// TIA Portal V17 export
// export: Created 2025-03-05T08:01:38.605309Z, ExportSetting WithDefaults, DisplayName Totally Integrated Automation Portal, DisplayVersion V17 Update 8, DisplayName TIA Portal Openness, DisplayVersion V17 Update 8, DisplayName TIA Portal Version Control Interface, DisplayVersion V17, DisplayName SINAMICS Startdrive Advanced, DisplayVersion V17 SP2, DisplayName SINAMICS Startdrive G110M, G120, G120C, G120D, G120P, G115D, DisplayVersion V17 SP2, DisplayName SINAMICS Startdrive G130, G150, S120, S150, SINAMICS MV, S210, DisplayVersion V17 SP2, DisplayName STEP 7 Professional, DisplayVersion V17 Update 8, DisplayName SINUMERIK ONE STEP 7 Toolbox, DisplayVersion V17 Update 12, DisplayName SINUMERIK 840D sl STEP 7 Toolbox, DisplayVersion V17 Update 12, DisplayName STEP 7 Safety, DisplayVersion V17 Update 6, DisplayName WinCC Advanced, DisplayVersion V17 Update 8
FUNCTION "FC7217_TRADES_CALL" : Void   // FC7217, LAD
{ S7_Optimized_Access := 'FALSE' }
AUTHOR : ETXETAR
VERSION : 1.0
// stored: AutoNumber false, IsIECCheckEnabled false, SetENOAutomatically false, UDAEnableTagReadback false
   VAR CONSTANT
      FC_NUMBER : DInt := 7217;
   END_VAR
   VAR_TEMP   // added for the SCL form of the ladder/FBD networks
      _w1 : Bool;
      _w2 : Bool;
      _w3 : Bool;
      _w4 : Bool;
      _w5 : Bool;
      _w6 : Bool;
      _w7 : Bool;
      _w8 : Bool;
      _w9 : Bool;
      _w10 : Bool;
      _w11 : Bool;
      _w12 : Bool;
      _w13 : Bool;
      _w14 : Bool;
      _w15 : Bool;
      _w16 : Bool;
   END_VAR
BEGIN

REGION Network 1: GENERAL CONDITIONS
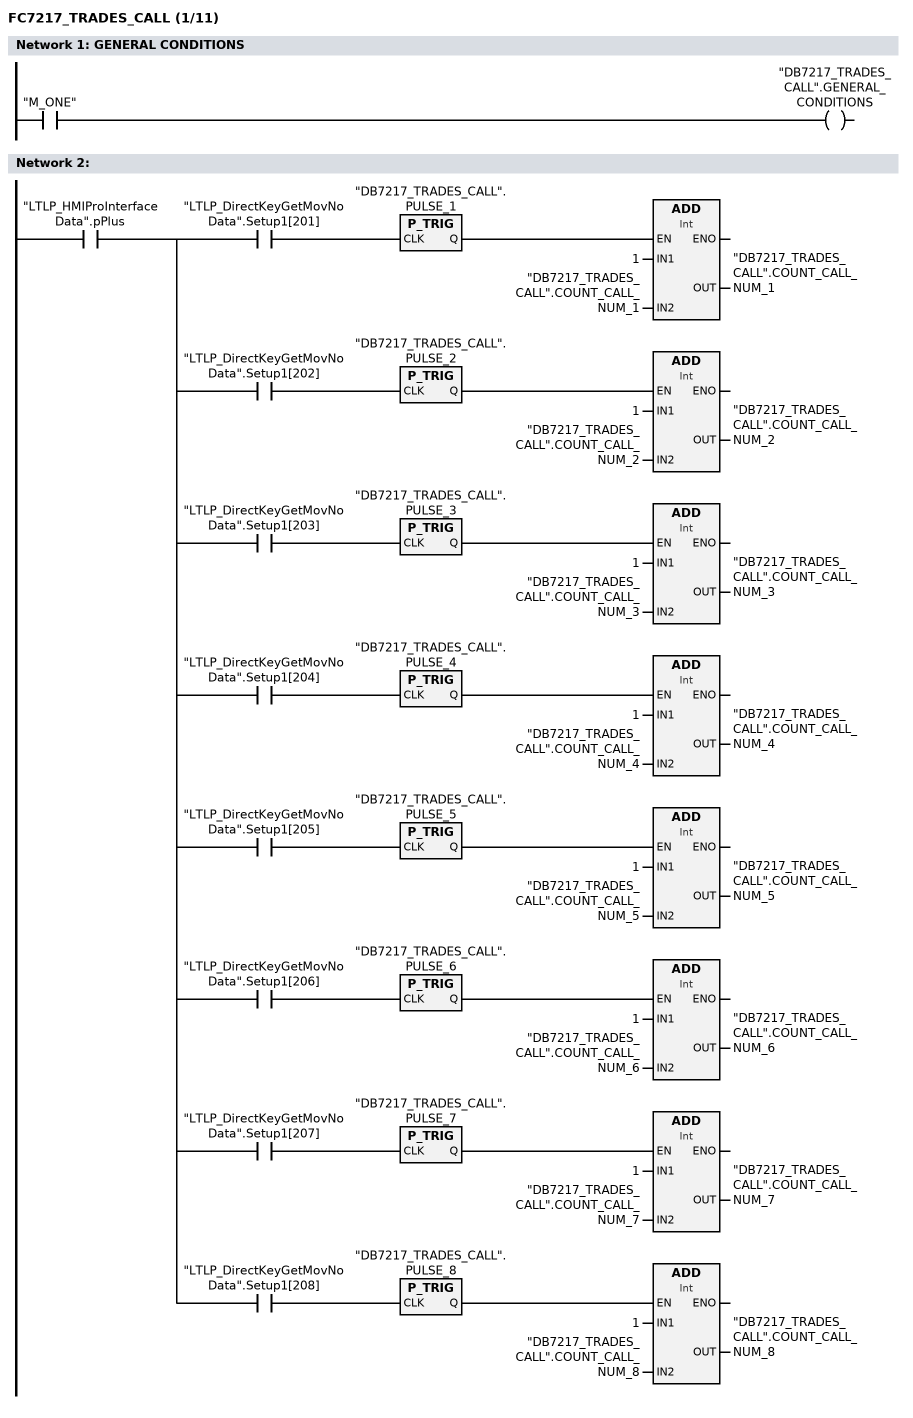
   RUNG wire#powerrail
      Contact( "M_ONE" )
      Coil( "DB7217_TRADES_CALL".GENERAL_CONDITIONS )
   END_RUNG
   // the same network as SCL:
   "DB7217_TRADES_CALL".GENERAL_CONDITIONS := "M_ONE";
END_REGION

REGION Network 2
   RUNG wire#powerrail
      Contact( "LTLP_HMIProInterfaceData".pPlus )
      wire#w1
      Contact( "LTLP_DirectKeyGetMovNoData".Setup1[201] )
      P_Trig( "DB7217_TRADES_CALL".PULSE_1 )
      { S7_Templates := "SrcType := Int"; S7_GenerateENO := "TRUE" } Add(in1 := 1, in2 := "DB7217_TRADES_CALL".COUNT_CALL_NUM_1, out => "DB7217_TRADES_CALL".COUNT_CALL_NUM_1)
   END_RUNG
   RUNG wire#w1
      Contact( "LTLP_DirectKeyGetMovNoData".Setup1[202] )
      P_Trig( "DB7217_TRADES_CALL".PULSE_2 )
      { S7_Templates := "SrcType := Int"; S7_GenerateENO := "TRUE" } Add(in1 := 1, in2 := "DB7217_TRADES_CALL".COUNT_CALL_NUM_2, out => "DB7217_TRADES_CALL".COUNT_CALL_NUM_2)
   END_RUNG
   RUNG wire#w1
      Contact( "LTLP_DirectKeyGetMovNoData".Setup1[203] )
      P_Trig( "DB7217_TRADES_CALL".PULSE_3 )
      { S7_Templates := "SrcType := Int"; S7_GenerateENO := "TRUE" } Add(in1 := 1, in2 := "DB7217_TRADES_CALL".COUNT_CALL_NUM_3, out => "DB7217_TRADES_CALL".COUNT_CALL_NUM_3)
   END_RUNG
   RUNG wire#w1
      Contact( "LTLP_DirectKeyGetMovNoData".Setup1[204] )
      P_Trig( "DB7217_TRADES_CALL".PULSE_4 )
      { S7_Templates := "SrcType := Int"; S7_GenerateENO := "TRUE" } Add(in1 := 1, in2 := "DB7217_TRADES_CALL".COUNT_CALL_NUM_4, out => "DB7217_TRADES_CALL".COUNT_CALL_NUM_4)
   END_RUNG
   RUNG wire#w1
      Contact( "LTLP_DirectKeyGetMovNoData".Setup1[205] )
      P_Trig( "DB7217_TRADES_CALL".PULSE_5 )
      { S7_Templates := "SrcType := Int"; S7_GenerateENO := "TRUE" } Add(in1 := 1, in2 := "DB7217_TRADES_CALL".COUNT_CALL_NUM_5, out => "DB7217_TRADES_CALL".COUNT_CALL_NUM_5)
   END_RUNG
   RUNG wire#w1
      Contact( "LTLP_DirectKeyGetMovNoData".Setup1[206] )
      P_Trig( "DB7217_TRADES_CALL".PULSE_6 )
      { S7_Templates := "SrcType := Int"; S7_GenerateENO := "TRUE" } Add(in1 := 1, in2 := "DB7217_TRADES_CALL".COUNT_CALL_NUM_6, out => "DB7217_TRADES_CALL".COUNT_CALL_NUM_6)
   END_RUNG
   RUNG wire#w1
      Contact( "LTLP_DirectKeyGetMovNoData".Setup1[207] )
      P_Trig( "DB7217_TRADES_CALL".PULSE_7 )
      { S7_Templates := "SrcType := Int"; S7_GenerateENO := "TRUE" } Add(in1 := 1, in2 := "DB7217_TRADES_CALL".COUNT_CALL_NUM_7, out => "DB7217_TRADES_CALL".COUNT_CALL_NUM_7)
   END_RUNG
   RUNG wire#w1
      Contact( "LTLP_DirectKeyGetMovNoData".Setup1[208] )
      P_Trig( "DB7217_TRADES_CALL".PULSE_8 )
      { S7_Templates := "SrcType := Int"; S7_GenerateENO := "TRUE" } Add(in1 := 1, in2 := "DB7217_TRADES_CALL".COUNT_CALL_NUM_8, out => "DB7217_TRADES_CALL".COUNT_CALL_NUM_8)
   END_RUNG
   // the same network as SCL:
   #_w1 := "LTLP_HMIProInterfaceData".pPlus AND "LTLP_DirectKeyGetMovNoData".Setup1[201];
   #_w2 := #_w1 AND NOT "DB7217_TRADES_CALL".PULSE_1;   // rising edge
   "DB7217_TRADES_CALL".PULSE_1 := #_w1;
   IF #_w2 THEN "DB7217_TRADES_CALL".COUNT_CALL_NUM_1 := 1 + "DB7217_TRADES_CALL".COUNT_CALL_NUM_1; END_IF;
   #_w3 := "LTLP_HMIProInterfaceData".pPlus AND "LTLP_DirectKeyGetMovNoData".Setup1[202];
   #_w4 := #_w3 AND NOT "DB7217_TRADES_CALL".PULSE_2;   // rising edge
   "DB7217_TRADES_CALL".PULSE_2 := #_w3;
   IF #_w4 THEN "DB7217_TRADES_CALL".COUNT_CALL_NUM_2 := 1 + "DB7217_TRADES_CALL".COUNT_CALL_NUM_2; END_IF;
   #_w5 := "LTLP_HMIProInterfaceData".pPlus AND "LTLP_DirectKeyGetMovNoData".Setup1[203];
   #_w6 := #_w5 AND NOT "DB7217_TRADES_CALL".PULSE_3;   // rising edge
   "DB7217_TRADES_CALL".PULSE_3 := #_w5;
   IF #_w6 THEN "DB7217_TRADES_CALL".COUNT_CALL_NUM_3 := 1 + "DB7217_TRADES_CALL".COUNT_CALL_NUM_3; END_IF;
   #_w7 := "LTLP_HMIProInterfaceData".pPlus AND "LTLP_DirectKeyGetMovNoData".Setup1[204];
   #_w8 := #_w7 AND NOT "DB7217_TRADES_CALL".PULSE_4;   // rising edge
   "DB7217_TRADES_CALL".PULSE_4 := #_w7;
   IF #_w8 THEN "DB7217_TRADES_CALL".COUNT_CALL_NUM_4 := 1 + "DB7217_TRADES_CALL".COUNT_CALL_NUM_4; END_IF;
   #_w9 := "LTLP_HMIProInterfaceData".pPlus AND "LTLP_DirectKeyGetMovNoData".Setup1[205];
   #_w10 := #_w9 AND NOT "DB7217_TRADES_CALL".PULSE_5;   // rising edge
   "DB7217_TRADES_CALL".PULSE_5 := #_w9;
   IF #_w10 THEN "DB7217_TRADES_CALL".COUNT_CALL_NUM_5 := 1 + "DB7217_TRADES_CALL".COUNT_CALL_NUM_5; END_IF;
   #_w11 := "LTLP_HMIProInterfaceData".pPlus AND "LTLP_DirectKeyGetMovNoData".Setup1[206];
   #_w12 := #_w11 AND NOT "DB7217_TRADES_CALL".PULSE_6;   // rising edge
   "DB7217_TRADES_CALL".PULSE_6 := #_w11;
   IF #_w12 THEN "DB7217_TRADES_CALL".COUNT_CALL_NUM_6 := 1 + "DB7217_TRADES_CALL".COUNT_CALL_NUM_6; END_IF;
   #_w13 := "LTLP_HMIProInterfaceData".pPlus AND "LTLP_DirectKeyGetMovNoData".Setup1[207];
   #_w14 := #_w13 AND NOT "DB7217_TRADES_CALL".PULSE_7;   // rising edge
   "DB7217_TRADES_CALL".PULSE_7 := #_w13;
   IF #_w14 THEN "DB7217_TRADES_CALL".COUNT_CALL_NUM_7 := 1 + "DB7217_TRADES_CALL".COUNT_CALL_NUM_7; END_IF;
   #_w15 := "LTLP_HMIProInterfaceData".pPlus AND "LTLP_DirectKeyGetMovNoData".Setup1[208];
   #_w16 := #_w15 AND NOT "DB7217_TRADES_CALL".PULSE_8;   // rising edge
   "DB7217_TRADES_CALL".PULSE_8 := #_w15;
   IF #_w16 THEN "DB7217_TRADES_CALL".COUNT_CALL_NUM_8 := 1 + "DB7217_TRADES_CALL".COUNT_CALL_NUM_8; END_IF;
END_REGION

REGION Network 3: CALL 1 AUX
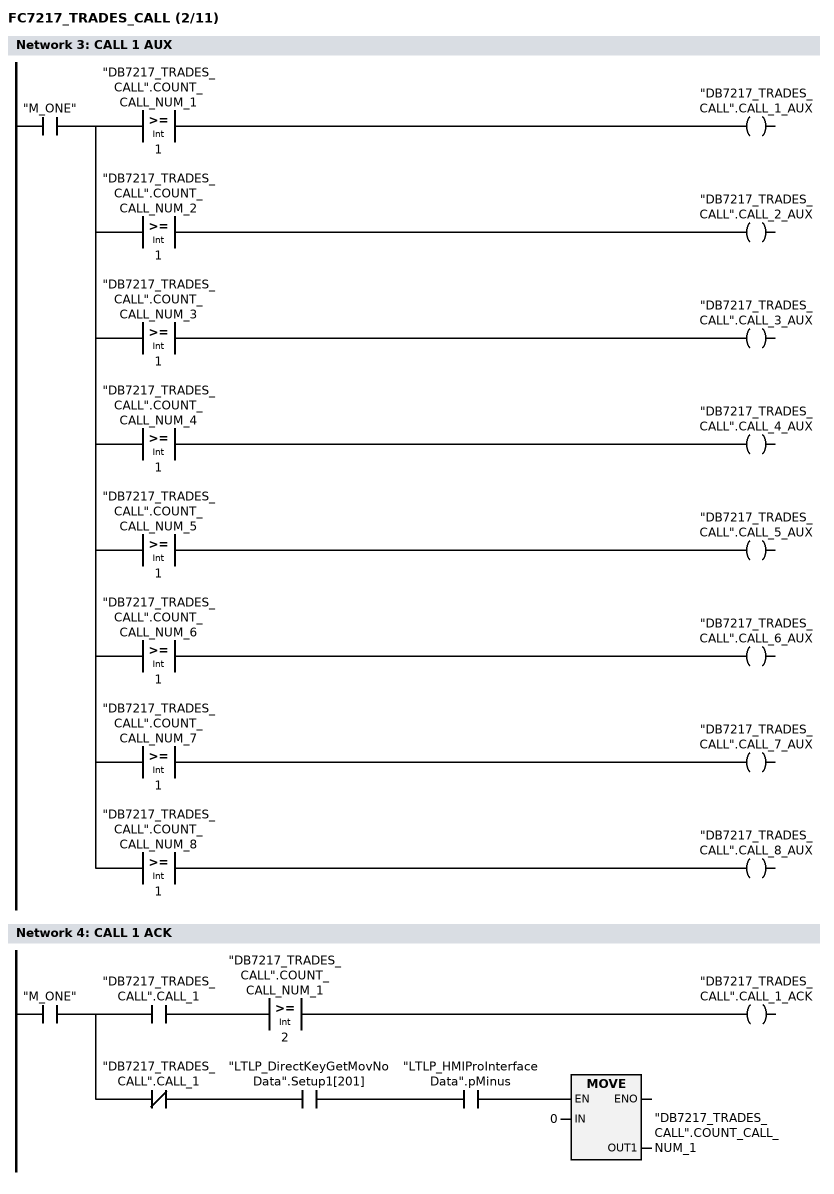
   RUNG wire#powerrail
      Contact( "M_ONE" )
      wire#w1
      { S7_Templates := "SrcType := Int" } GE_Contact(in1 := "DB7217_TRADES_CALL".COUNT_CALL_NUM_1, in2 := 1)
      Coil( "DB7217_TRADES_CALL".CALL_1_AUX )
   END_RUNG
   RUNG wire#w1
      { S7_Templates := "SrcType := Int" } GE_Contact(in1 := "DB7217_TRADES_CALL".COUNT_CALL_NUM_2, in2 := 1)
      Coil( "DB7217_TRADES_CALL".CALL_2_AUX )
   END_RUNG
   RUNG wire#w1
      { S7_Templates := "SrcType := Int" } GE_Contact(in1 := "DB7217_TRADES_CALL".COUNT_CALL_NUM_3, in2 := 1)
      Coil( "DB7217_TRADES_CALL".CALL_3_AUX )
   END_RUNG
   RUNG wire#w1
      { S7_Templates := "SrcType := Int" } GE_Contact(in1 := "DB7217_TRADES_CALL".COUNT_CALL_NUM_4, in2 := 1)
      Coil( "DB7217_TRADES_CALL".CALL_4_AUX )
   END_RUNG
   RUNG wire#w1
      { S7_Templates := "SrcType := Int" } GE_Contact(in1 := "DB7217_TRADES_CALL".COUNT_CALL_NUM_5, in2 := 1)
      Coil( "DB7217_TRADES_CALL".CALL_5_AUX )
   END_RUNG
   RUNG wire#w1
      { S7_Templates := "SrcType := Int" } GE_Contact(in1 := "DB7217_TRADES_CALL".COUNT_CALL_NUM_6, in2 := 1)
      Coil( "DB7217_TRADES_CALL".CALL_6_AUX )
   END_RUNG
   RUNG wire#w1
      { S7_Templates := "SrcType := Int" } GE_Contact(in1 := "DB7217_TRADES_CALL".COUNT_CALL_NUM_7, in2 := 1)
      Coil( "DB7217_TRADES_CALL".CALL_7_AUX )
   END_RUNG
   RUNG wire#w1
      { S7_Templates := "SrcType := Int" } GE_Contact(in1 := "DB7217_TRADES_CALL".COUNT_CALL_NUM_8, in2 := 1)
      Coil( "DB7217_TRADES_CALL".CALL_8_AUX )
   END_RUNG
   // the same network as SCL:
   "DB7217_TRADES_CALL".CALL_1_AUX := "M_ONE" AND ("DB7217_TRADES_CALL".COUNT_CALL_NUM_1 >= 1);
   "DB7217_TRADES_CALL".CALL_2_AUX := "M_ONE" AND ("DB7217_TRADES_CALL".COUNT_CALL_NUM_2 >= 1);
   "DB7217_TRADES_CALL".CALL_3_AUX := "M_ONE" AND ("DB7217_TRADES_CALL".COUNT_CALL_NUM_3 >= 1);
   "DB7217_TRADES_CALL".CALL_4_AUX := "M_ONE" AND ("DB7217_TRADES_CALL".COUNT_CALL_NUM_4 >= 1);
   "DB7217_TRADES_CALL".CALL_5_AUX := "M_ONE" AND ("DB7217_TRADES_CALL".COUNT_CALL_NUM_5 >= 1);
   "DB7217_TRADES_CALL".CALL_6_AUX := "M_ONE" AND ("DB7217_TRADES_CALL".COUNT_CALL_NUM_6 >= 1);
   "DB7217_TRADES_CALL".CALL_7_AUX := "M_ONE" AND ("DB7217_TRADES_CALL".COUNT_CALL_NUM_7 >= 1);
   "DB7217_TRADES_CALL".CALL_8_AUX := "M_ONE" AND ("DB7217_TRADES_CALL".COUNT_CALL_NUM_8 >= 1);
END_REGION

REGION Network 4: CALL 1 ACK
   RUNG wire#powerrail
      Contact( "M_ONE" )
      wire#w1
      Contact( "DB7217_TRADES_CALL".CALL_1 )
      { S7_Templates := "SrcType := Int" } GE_Contact(in1 := "DB7217_TRADES_CALL".COUNT_CALL_NUM_1, in2 := 2)
      Coil( "DB7217_TRADES_CALL".CALL_1_ACK )
   END_RUNG
   RUNG wire#w1
      I_Contact( "DB7217_TRADES_CALL".CALL_1 )
      Contact( "LTLP_DirectKeyGetMovNoData".Setup1[201] )
      Contact( "LTLP_HMIProInterfaceData".pMinus )
      { S7_GenerateENO := "TRUE" } Move(in := 0, out1 => "DB7217_TRADES_CALL".COUNT_CALL_NUM_1)
   END_RUNG
   // the same network as SCL:
   "DB7217_TRADES_CALL".CALL_1_ACK := "M_ONE" AND "DB7217_TRADES_CALL".CALL_1 AND ("DB7217_TRADES_CALL".COUNT_CALL_NUM_1 >= 2);
   IF "M_ONE" AND NOT "DB7217_TRADES_CALL".CALL_1 AND "LTLP_DirectKeyGetMovNoData".Setup1[201] AND "LTLP_HMIProInterfaceData".pMinus THEN
       "DB7217_TRADES_CALL".COUNT_CALL_NUM_1 := 0;
   END_IF;
END_REGION

REGION Network 5: CALL 2 ACK
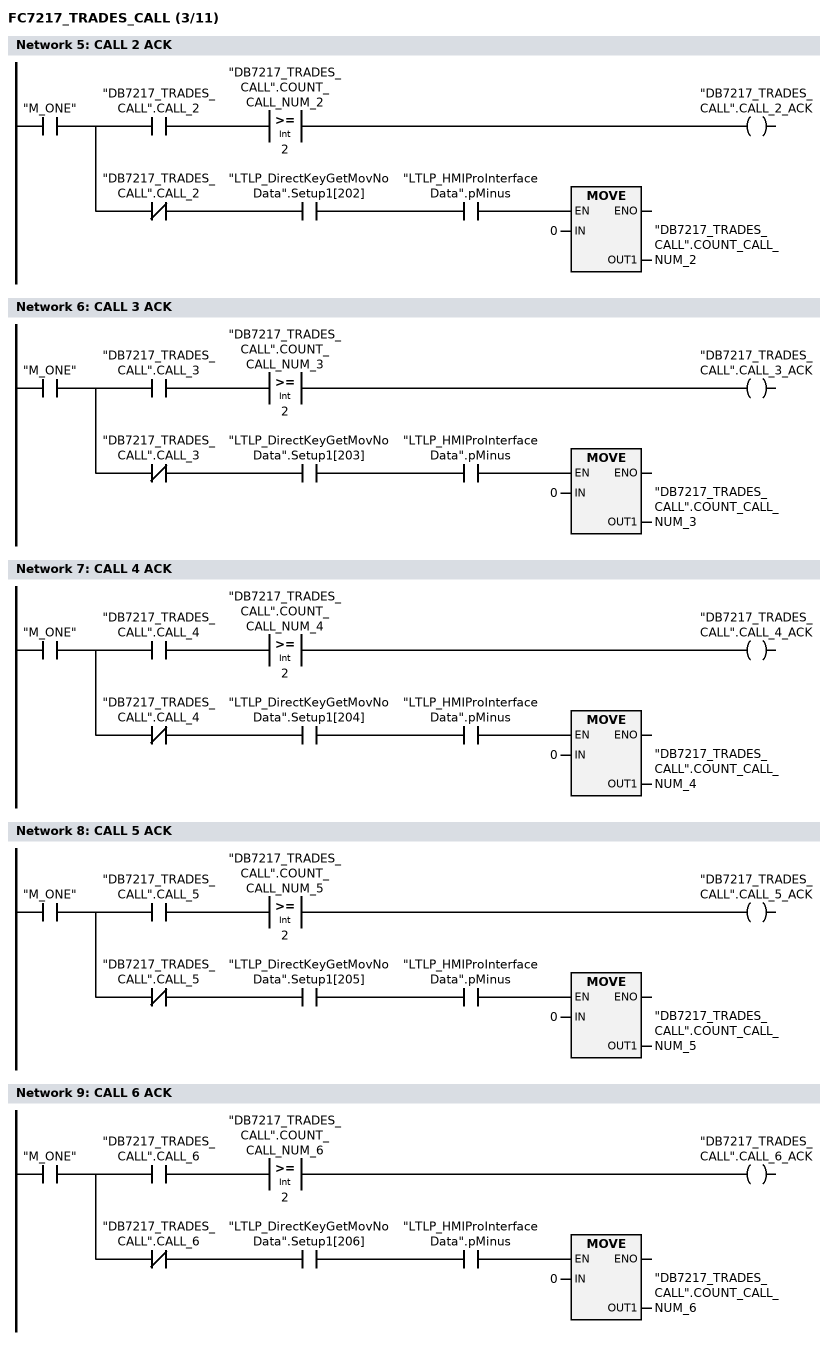
   RUNG wire#powerrail
      Contact( "M_ONE" )
      wire#w1
      Contact( "DB7217_TRADES_CALL".CALL_2 )
      { S7_Templates := "SrcType := Int" } GE_Contact(in1 := "DB7217_TRADES_CALL".COUNT_CALL_NUM_2, in2 := 2)
      Coil( "DB7217_TRADES_CALL".CALL_2_ACK )
   END_RUNG
   RUNG wire#w1
      I_Contact( "DB7217_TRADES_CALL".CALL_2 )
      Contact( "LTLP_DirectKeyGetMovNoData".Setup1[202] )
      Contact( "LTLP_HMIProInterfaceData".pMinus )
      { S7_GenerateENO := "TRUE" } Move(in := 0, out1 => "DB7217_TRADES_CALL".COUNT_CALL_NUM_2)
   END_RUNG
   // the same network as SCL:
   "DB7217_TRADES_CALL".CALL_2_ACK := "M_ONE" AND "DB7217_TRADES_CALL".CALL_2 AND ("DB7217_TRADES_CALL".COUNT_CALL_NUM_2 >= 2);
   IF "M_ONE" AND NOT "DB7217_TRADES_CALL".CALL_2 AND "LTLP_DirectKeyGetMovNoData".Setup1[202] AND "LTLP_HMIProInterfaceData".pMinus THEN
       "DB7217_TRADES_CALL".COUNT_CALL_NUM_2 := 0;
   END_IF;
END_REGION

REGION Network 6: CALL 3 ACK
   RUNG wire#powerrail
      Contact( "M_ONE" )
      wire#w1
      Contact( "DB7217_TRADES_CALL".CALL_3 )
      { S7_Templates := "SrcType := Int" } GE_Contact(in1 := "DB7217_TRADES_CALL".COUNT_CALL_NUM_3, in2 := 2)
      Coil( "DB7217_TRADES_CALL".CALL_3_ACK )
   END_RUNG
   RUNG wire#w1
      I_Contact( "DB7217_TRADES_CALL".CALL_3 )
      Contact( "LTLP_DirectKeyGetMovNoData".Setup1[203] )
      Contact( "LTLP_HMIProInterfaceData".pMinus )
      { S7_GenerateENO := "TRUE" } Move(in := 0, out1 => "DB7217_TRADES_CALL".COUNT_CALL_NUM_3)
   END_RUNG
   // the same network as SCL:
   "DB7217_TRADES_CALL".CALL_3_ACK := "M_ONE" AND "DB7217_TRADES_CALL".CALL_3 AND ("DB7217_TRADES_CALL".COUNT_CALL_NUM_3 >= 2);
   IF "M_ONE" AND NOT "DB7217_TRADES_CALL".CALL_3 AND "LTLP_DirectKeyGetMovNoData".Setup1[203] AND "LTLP_HMIProInterfaceData".pMinus THEN
       "DB7217_TRADES_CALL".COUNT_CALL_NUM_3 := 0;
   END_IF;
END_REGION

REGION Network 7: CALL 4 ACK
   RUNG wire#powerrail
      Contact( "M_ONE" )
      wire#w1
      Contact( "DB7217_TRADES_CALL".CALL_4 )
      { S7_Templates := "SrcType := Int" } GE_Contact(in1 := "DB7217_TRADES_CALL".COUNT_CALL_NUM_4, in2 := 2)
      Coil( "DB7217_TRADES_CALL".CALL_4_ACK )
   END_RUNG
   RUNG wire#w1
      I_Contact( "DB7217_TRADES_CALL".CALL_4 )
      Contact( "LTLP_DirectKeyGetMovNoData".Setup1[204] )
      Contact( "LTLP_HMIProInterfaceData".pMinus )
      { S7_GenerateENO := "TRUE" } Move(in := 0, out1 => "DB7217_TRADES_CALL".COUNT_CALL_NUM_4)
   END_RUNG
   // the same network as SCL:
   "DB7217_TRADES_CALL".CALL_4_ACK := "M_ONE" AND "DB7217_TRADES_CALL".CALL_4 AND ("DB7217_TRADES_CALL".COUNT_CALL_NUM_4 >= 2);
   IF "M_ONE" AND NOT "DB7217_TRADES_CALL".CALL_4 AND "LTLP_DirectKeyGetMovNoData".Setup1[204] AND "LTLP_HMIProInterfaceData".pMinus THEN
       "DB7217_TRADES_CALL".COUNT_CALL_NUM_4 := 0;
   END_IF;
END_REGION

REGION Network 8: CALL 5 ACK
   RUNG wire#powerrail
      Contact( "M_ONE" )
      wire#w1
      Contact( "DB7217_TRADES_CALL".CALL_5 )
      { S7_Templates := "SrcType := Int" } GE_Contact(in1 := "DB7217_TRADES_CALL".COUNT_CALL_NUM_5, in2 := 2)
      Coil( "DB7217_TRADES_CALL".CALL_5_ACK )
   END_RUNG
   RUNG wire#w1
      I_Contact( "DB7217_TRADES_CALL".CALL_5 )
      Contact( "LTLP_DirectKeyGetMovNoData".Setup1[205] )
      Contact( "LTLP_HMIProInterfaceData".pMinus )
      { S7_GenerateENO := "TRUE" } Move(in := 0, out1 => "DB7217_TRADES_CALL".COUNT_CALL_NUM_5)
   END_RUNG
   // the same network as SCL:
   "DB7217_TRADES_CALL".CALL_5_ACK := "M_ONE" AND "DB7217_TRADES_CALL".CALL_5 AND ("DB7217_TRADES_CALL".COUNT_CALL_NUM_5 >= 2);
   IF "M_ONE" AND NOT "DB7217_TRADES_CALL".CALL_5 AND "LTLP_DirectKeyGetMovNoData".Setup1[205] AND "LTLP_HMIProInterfaceData".pMinus THEN
       "DB7217_TRADES_CALL".COUNT_CALL_NUM_5 := 0;
   END_IF;
END_REGION

REGION Network 9: CALL 6 ACK
   RUNG wire#powerrail
      Contact( "M_ONE" )
      wire#w1
      Contact( "DB7217_TRADES_CALL".CALL_6 )
      { S7_Templates := "SrcType := Int" } GE_Contact(in1 := "DB7217_TRADES_CALL".COUNT_CALL_NUM_6, in2 := 2)
      Coil( "DB7217_TRADES_CALL".CALL_6_ACK )
   END_RUNG
   RUNG wire#w1
      I_Contact( "DB7217_TRADES_CALL".CALL_6 )
      Contact( "LTLP_DirectKeyGetMovNoData".Setup1[206] )
      Contact( "LTLP_HMIProInterfaceData".pMinus )
      { S7_GenerateENO := "TRUE" } Move(in := 0, out1 => "DB7217_TRADES_CALL".COUNT_CALL_NUM_6)
   END_RUNG
   // the same network as SCL:
   "DB7217_TRADES_CALL".CALL_6_ACK := "M_ONE" AND "DB7217_TRADES_CALL".CALL_6 AND ("DB7217_TRADES_CALL".COUNT_CALL_NUM_6 >= 2);
   IF "M_ONE" AND NOT "DB7217_TRADES_CALL".CALL_6 AND "LTLP_DirectKeyGetMovNoData".Setup1[206] AND "LTLP_HMIProInterfaceData".pMinus THEN
       "DB7217_TRADES_CALL".COUNT_CALL_NUM_6 := 0;
   END_IF;
END_REGION

REGION Network 10: CALL 7 ACK
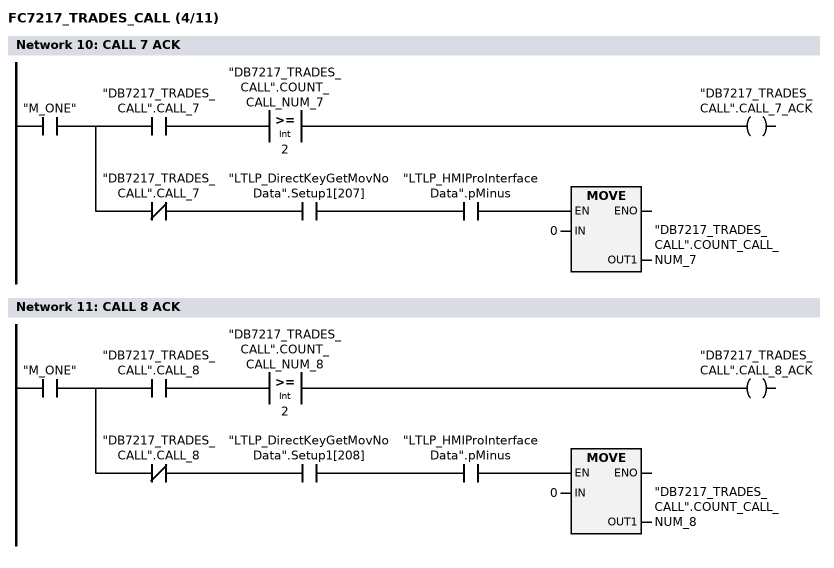
   RUNG wire#powerrail
      Contact( "M_ONE" )
      wire#w1
      Contact( "DB7217_TRADES_CALL".CALL_7 )
      { S7_Templates := "SrcType := Int" } GE_Contact(in1 := "DB7217_TRADES_CALL".COUNT_CALL_NUM_7, in2 := 2)
      Coil( "DB7217_TRADES_CALL".CALL_7_ACK )
   END_RUNG
   RUNG wire#w1
      I_Contact( "DB7217_TRADES_CALL".CALL_7 )
      Contact( "LTLP_DirectKeyGetMovNoData".Setup1[207] )
      Contact( "LTLP_HMIProInterfaceData".pMinus )
      { S7_GenerateENO := "TRUE" } Move(in := 0, out1 => "DB7217_TRADES_CALL".COUNT_CALL_NUM_7)
   END_RUNG
   // the same network as SCL:
   "DB7217_TRADES_CALL".CALL_7_ACK := "M_ONE" AND "DB7217_TRADES_CALL".CALL_7 AND ("DB7217_TRADES_CALL".COUNT_CALL_NUM_7 >= 2);
   IF "M_ONE" AND NOT "DB7217_TRADES_CALL".CALL_7 AND "LTLP_DirectKeyGetMovNoData".Setup1[207] AND "LTLP_HMIProInterfaceData".pMinus THEN
       "DB7217_TRADES_CALL".COUNT_CALL_NUM_7 := 0;
   END_IF;
END_REGION

REGION Network 11: CALL 8 ACK
   RUNG wire#powerrail
      Contact( "M_ONE" )
      wire#w1
      Contact( "DB7217_TRADES_CALL".CALL_8 )
      { S7_Templates := "SrcType := Int" } GE_Contact(in1 := "DB7217_TRADES_CALL".COUNT_CALL_NUM_8, in2 := 2)
      Coil( "DB7217_TRADES_CALL".CALL_8_ACK )
   END_RUNG
   RUNG wire#w1
      I_Contact( "DB7217_TRADES_CALL".CALL_8 )
      Contact( "LTLP_DirectKeyGetMovNoData".Setup1[208] )
      Contact( "LTLP_HMIProInterfaceData".pMinus )
      { S7_GenerateENO := "TRUE" } Move(in := 0, out1 => "DB7217_TRADES_CALL".COUNT_CALL_NUM_8)
   END_RUNG
   // the same network as SCL:
   "DB7217_TRADES_CALL".CALL_8_ACK := "M_ONE" AND "DB7217_TRADES_CALL".CALL_8 AND ("DB7217_TRADES_CALL".COUNT_CALL_NUM_8 >= 2);
   IF "M_ONE" AND NOT "DB7217_TRADES_CALL".CALL_8 AND "LTLP_DirectKeyGetMovNoData".Setup1[208] AND "LTLP_HMIProInterfaceData".pMinus THEN
       "DB7217_TRADES_CALL".COUNT_CALL_NUM_8 := 0;
   END_IF;
END_REGION

REGION Network 12: CALL 1 REQ
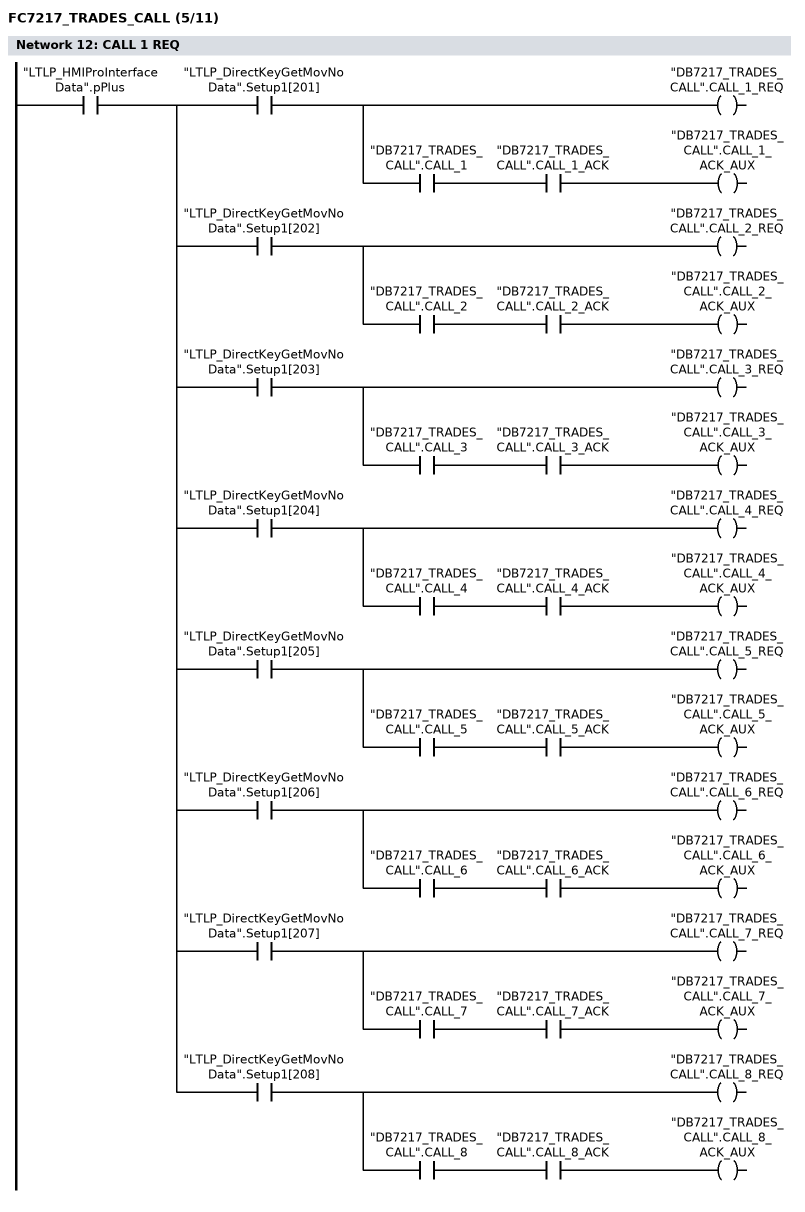
   RUNG wire#powerrail
      Contact( "LTLP_HMIProInterfaceData".pPlus )
      wire#w1
      Contact( "LTLP_DirectKeyGetMovNoData".Setup1[201] )
      wire#w2
      Coil( "DB7217_TRADES_CALL".CALL_1_REQ )
   END_RUNG
   RUNG wire#w2
      Contact( "DB7217_TRADES_CALL".CALL_1 )
      Contact( "DB7217_TRADES_CALL".CALL_1_ACK )
      Coil( "DB7217_TRADES_CALL".CALL_1_ACK_AUX )
   END_RUNG
   RUNG wire#w1
      Contact( "LTLP_DirectKeyGetMovNoData".Setup1[202] )
      wire#w3
      Coil( "DB7217_TRADES_CALL".CALL_2_REQ )
   END_RUNG
   RUNG wire#w3
      Contact( "DB7217_TRADES_CALL".CALL_2 )
      Contact( "DB7217_TRADES_CALL".CALL_2_ACK )
      Coil( "DB7217_TRADES_CALL".CALL_2_ACK_AUX )
   END_RUNG
   RUNG wire#w1
      Contact( "LTLP_DirectKeyGetMovNoData".Setup1[203] )
      wire#w4
      Coil( "DB7217_TRADES_CALL".CALL_3_REQ )
   END_RUNG
   RUNG wire#w4
      Contact( "DB7217_TRADES_CALL".CALL_3 )
      Contact( "DB7217_TRADES_CALL".CALL_3_ACK )
      Coil( "DB7217_TRADES_CALL".CALL_3_ACK_AUX )
   END_RUNG
   RUNG wire#w1
      Contact( "LTLP_DirectKeyGetMovNoData".Setup1[204] )
      wire#w5
      Coil( "DB7217_TRADES_CALL".CALL_4_REQ )
   END_RUNG
   RUNG wire#w5
      Contact( "DB7217_TRADES_CALL".CALL_4 )
      Contact( "DB7217_TRADES_CALL".CALL_4_ACK )
      Coil( "DB7217_TRADES_CALL".CALL_4_ACK_AUX )
   END_RUNG
   RUNG wire#w1
      Contact( "LTLP_DirectKeyGetMovNoData".Setup1[205] )
      wire#w6
      Coil( "DB7217_TRADES_CALL".CALL_5_REQ )
   END_RUNG
   RUNG wire#w6
      Contact( "DB7217_TRADES_CALL".CALL_5 )
      Contact( "DB7217_TRADES_CALL".CALL_5_ACK )
      Coil( "DB7217_TRADES_CALL".CALL_5_ACK_AUX )
   END_RUNG
   RUNG wire#w1
      Contact( "LTLP_DirectKeyGetMovNoData".Setup1[206] )
      wire#w7
      Coil( "DB7217_TRADES_CALL".CALL_6_REQ )
   END_RUNG
   RUNG wire#w7
      Contact( "DB7217_TRADES_CALL".CALL_6 )
      Contact( "DB7217_TRADES_CALL".CALL_6_ACK )
      Coil( "DB7217_TRADES_CALL".CALL_6_ACK_AUX )
   END_RUNG
   RUNG wire#w1
      Contact( "LTLP_DirectKeyGetMovNoData".Setup1[207] )
      wire#w8
      Coil( "DB7217_TRADES_CALL".CALL_7_REQ )
   END_RUNG
   RUNG wire#w8
      Contact( "DB7217_TRADES_CALL".CALL_7 )
      Contact( "DB7217_TRADES_CALL".CALL_7_ACK )
      Coil( "DB7217_TRADES_CALL".CALL_7_ACK_AUX )
   END_RUNG
   RUNG wire#w1
      Contact( "LTLP_DirectKeyGetMovNoData".Setup1[208] )
      wire#w9
      Coil( "DB7217_TRADES_CALL".CALL_8_REQ )
   END_RUNG
   RUNG wire#w9
      Contact( "DB7217_TRADES_CALL".CALL_8 )
      Contact( "DB7217_TRADES_CALL".CALL_8_ACK )
      Coil( "DB7217_TRADES_CALL".CALL_8_ACK_AUX )
   END_RUNG
   // the same network as SCL:
   "DB7217_TRADES_CALL".CALL_1_REQ := "LTLP_HMIProInterfaceData".pPlus AND "LTLP_DirectKeyGetMovNoData".Setup1[201];
   "DB7217_TRADES_CALL".CALL_1_ACK_AUX := "DB7217_TRADES_CALL".CALL_1_REQ AND "DB7217_TRADES_CALL".CALL_1 AND "DB7217_TRADES_CALL".CALL_1_ACK;
   "DB7217_TRADES_CALL".CALL_2_REQ := "LTLP_HMIProInterfaceData".pPlus AND "LTLP_DirectKeyGetMovNoData".Setup1[202];
   "DB7217_TRADES_CALL".CALL_2_ACK_AUX := "DB7217_TRADES_CALL".CALL_2_REQ AND "DB7217_TRADES_CALL".CALL_2 AND "DB7217_TRADES_CALL".CALL_2_ACK;
   "DB7217_TRADES_CALL".CALL_3_REQ := "LTLP_HMIProInterfaceData".pPlus AND "LTLP_DirectKeyGetMovNoData".Setup1[203];
   "DB7217_TRADES_CALL".CALL_3_ACK_AUX := "DB7217_TRADES_CALL".CALL_3_REQ AND "DB7217_TRADES_CALL".CALL_3 AND "DB7217_TRADES_CALL".CALL_3_ACK;
   "DB7217_TRADES_CALL".CALL_4_REQ := "LTLP_HMIProInterfaceData".pPlus AND "LTLP_DirectKeyGetMovNoData".Setup1[204];
   "DB7217_TRADES_CALL".CALL_4_ACK_AUX := "DB7217_TRADES_CALL".CALL_4_REQ AND "DB7217_TRADES_CALL".CALL_4 AND "DB7217_TRADES_CALL".CALL_4_ACK;
   "DB7217_TRADES_CALL".CALL_5_REQ := "LTLP_HMIProInterfaceData".pPlus AND "LTLP_DirectKeyGetMovNoData".Setup1[205];
   "DB7217_TRADES_CALL".CALL_5_ACK_AUX := "DB7217_TRADES_CALL".CALL_5_REQ AND "DB7217_TRADES_CALL".CALL_5 AND "DB7217_TRADES_CALL".CALL_5_ACK;
   "DB7217_TRADES_CALL".CALL_6_REQ := "LTLP_HMIProInterfaceData".pPlus AND "LTLP_DirectKeyGetMovNoData".Setup1[206];
   "DB7217_TRADES_CALL".CALL_6_ACK_AUX := "DB7217_TRADES_CALL".CALL_6_REQ AND "DB7217_TRADES_CALL".CALL_6 AND "DB7217_TRADES_CALL".CALL_6_ACK;
   "DB7217_TRADES_CALL".CALL_7_REQ := "LTLP_HMIProInterfaceData".pPlus AND "LTLP_DirectKeyGetMovNoData".Setup1[207];
   "DB7217_TRADES_CALL".CALL_7_ACK_AUX := "DB7217_TRADES_CALL".CALL_7_REQ AND "DB7217_TRADES_CALL".CALL_7 AND "DB7217_TRADES_CALL".CALL_7_ACK;
   "DB7217_TRADES_CALL".CALL_8_REQ := "LTLP_HMIProInterfaceData".pPlus AND "LTLP_DirectKeyGetMovNoData".Setup1[208];
   "DB7217_TRADES_CALL".CALL_8_ACK_AUX := "DB7217_TRADES_CALL".CALL_8_REQ AND "DB7217_TRADES_CALL".CALL_8 AND "DB7217_TRADES_CALL".CALL_8_ACK;
END_REGION

REGION Network 13: CANCEL 1 REQ
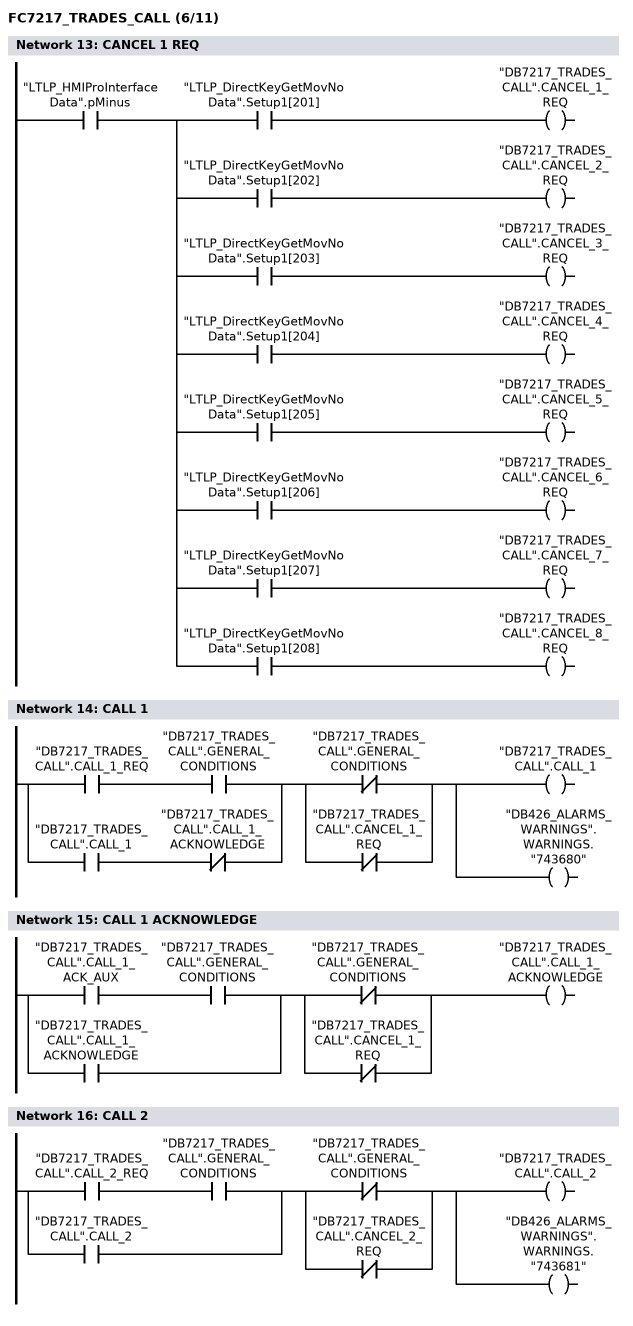
   RUNG wire#powerrail
      Contact( "LTLP_HMIProInterfaceData".pMinus )
      wire#w1
      Contact( "LTLP_DirectKeyGetMovNoData".Setup1[201] )
      Coil( "DB7217_TRADES_CALL".CANCEL_1_REQ )
   END_RUNG
   RUNG wire#w1
      Contact( "LTLP_DirectKeyGetMovNoData".Setup1[202] )
      Coil( "DB7217_TRADES_CALL".CANCEL_2_REQ )
   END_RUNG
   RUNG wire#w1
      Contact( "LTLP_DirectKeyGetMovNoData".Setup1[203] )
      Coil( "DB7217_TRADES_CALL".CANCEL_3_REQ )
   END_RUNG
   RUNG wire#w1
      Contact( "LTLP_DirectKeyGetMovNoData".Setup1[204] )
      Coil( "DB7217_TRADES_CALL".CANCEL_4_REQ )
   END_RUNG
   RUNG wire#w1
      Contact( "LTLP_DirectKeyGetMovNoData".Setup1[205] )
      Coil( "DB7217_TRADES_CALL".CANCEL_5_REQ )
   END_RUNG
   RUNG wire#w1
      Contact( "LTLP_DirectKeyGetMovNoData".Setup1[206] )
      Coil( "DB7217_TRADES_CALL".CANCEL_6_REQ )
   END_RUNG
   RUNG wire#w1
      Contact( "LTLP_DirectKeyGetMovNoData".Setup1[207] )
      Coil( "DB7217_TRADES_CALL".CANCEL_7_REQ )
   END_RUNG
   RUNG wire#w1
      Contact( "LTLP_DirectKeyGetMovNoData".Setup1[208] )
      Coil( "DB7217_TRADES_CALL".CANCEL_8_REQ )
   END_RUNG
   // the same network as SCL:
   "DB7217_TRADES_CALL".CANCEL_1_REQ := "LTLP_HMIProInterfaceData".pMinus AND "LTLP_DirectKeyGetMovNoData".Setup1[201];
   "DB7217_TRADES_CALL".CANCEL_2_REQ := "LTLP_HMIProInterfaceData".pMinus AND "LTLP_DirectKeyGetMovNoData".Setup1[202];
   "DB7217_TRADES_CALL".CANCEL_3_REQ := "LTLP_HMIProInterfaceData".pMinus AND "LTLP_DirectKeyGetMovNoData".Setup1[203];
   "DB7217_TRADES_CALL".CANCEL_4_REQ := "LTLP_HMIProInterfaceData".pMinus AND "LTLP_DirectKeyGetMovNoData".Setup1[204];
   "DB7217_TRADES_CALL".CANCEL_5_REQ := "LTLP_HMIProInterfaceData".pMinus AND "LTLP_DirectKeyGetMovNoData".Setup1[205];
   "DB7217_TRADES_CALL".CANCEL_6_REQ := "LTLP_HMIProInterfaceData".pMinus AND "LTLP_DirectKeyGetMovNoData".Setup1[206];
   "DB7217_TRADES_CALL".CANCEL_7_REQ := "LTLP_HMIProInterfaceData".pMinus AND "LTLP_DirectKeyGetMovNoData".Setup1[207];
   "DB7217_TRADES_CALL".CANCEL_8_REQ := "LTLP_HMIProInterfaceData".pMinus AND "LTLP_DirectKeyGetMovNoData".Setup1[208];
END_REGION

REGION Network 14: CALL 1
   RUNG wire#powerrail
      Contact( "DB7217_TRADES_CALL".CALL_1_REQ )
      Contact( "DB7217_TRADES_CALL".GENERAL_CONDITIONS )
      wire#w1
      I_Contact( "DB7217_TRADES_CALL".GENERAL_CONDITIONS )
      wire#w2
      Coil( "DB7217_TRADES_CALL".CALL_1 )
   END_RUNG
   RUNG wire#powerrail
      Contact( "DB7217_TRADES_CALL".CALL_1 )
      I_Contact( "DB7217_TRADES_CALL".CALL_1_ACKNOWLEDGE )
   END_RUNG wire#w1
   RUNG wire#w1
      I_Contact( "DB7217_TRADES_CALL".CANCEL_1_REQ )
   END_RUNG wire#w2
   RUNG wire#w2
      Coil( "DB426_ALARMS_WARNINGS".WARNINGS."743680" )
   END_RUNG
   // the same network as SCL:
   "DB7217_TRADES_CALL".CALL_1 := (("DB7217_TRADES_CALL".CALL_1_REQ AND "DB7217_TRADES_CALL".GENERAL_CONDITIONS) OR ("DB7217_TRADES_CALL".CALL_1 AND NOT "DB7217_TRADES_CALL".CALL_1_ACKNOWLEDGE)) AND (NOT "DB7217_TRADES_CALL".GENERAL_CONDITIONS OR NOT "DB7217_TRADES_CALL".CANCEL_1_REQ);
   "DB426_ALARMS_WARNINGS".WARNINGS."743680" := "DB7217_TRADES_CALL".CALL_1;
END_REGION

REGION Network 15: CALL 1 ACKNOWLEDGE
   RUNG wire#powerrail
      Contact( "DB7217_TRADES_CALL".CALL_1_ACK_AUX )
      Contact( "DB7217_TRADES_CALL".GENERAL_CONDITIONS )
      wire#w1
      I_Contact( "DB7217_TRADES_CALL".GENERAL_CONDITIONS )
      wire#w2
      Coil( "DB7217_TRADES_CALL".CALL_1_ACKNOWLEDGE )
   END_RUNG
   RUNG wire#powerrail
      Contact( "DB7217_TRADES_CALL".CALL_1_ACKNOWLEDGE )
   END_RUNG wire#w1
   RUNG wire#w1
      I_Contact( "DB7217_TRADES_CALL".CANCEL_1_REQ )
   END_RUNG wire#w2
   // the same network as SCL:
   "DB7217_TRADES_CALL".CALL_1_ACKNOWLEDGE := (("DB7217_TRADES_CALL".CALL_1_ACK_AUX AND "DB7217_TRADES_CALL".GENERAL_CONDITIONS) OR "DB7217_TRADES_CALL".CALL_1_ACKNOWLEDGE) AND (NOT "DB7217_TRADES_CALL".GENERAL_CONDITIONS OR NOT "DB7217_TRADES_CALL".CANCEL_1_REQ);
END_REGION

REGION Network 16: CALL 2
   RUNG wire#powerrail
      Contact( "DB7217_TRADES_CALL".CALL_2_REQ )
      Contact( "DB7217_TRADES_CALL".GENERAL_CONDITIONS )
      wire#w1
      I_Contact( "DB7217_TRADES_CALL".GENERAL_CONDITIONS )
      wire#w2
      Coil( "DB7217_TRADES_CALL".CALL_2 )
   END_RUNG
   RUNG wire#powerrail
      Contact( "DB7217_TRADES_CALL".CALL_2 )
   END_RUNG wire#w1
   RUNG wire#w1
      I_Contact( "DB7217_TRADES_CALL".CANCEL_2_REQ )
   END_RUNG wire#w2
   RUNG wire#w2
      Coil( "DB426_ALARMS_WARNINGS".WARNINGS."743681" )
   END_RUNG
   // the same network as SCL:
   "DB7217_TRADES_CALL".CALL_2 := (("DB7217_TRADES_CALL".CALL_2_REQ AND "DB7217_TRADES_CALL".GENERAL_CONDITIONS) OR "DB7217_TRADES_CALL".CALL_2) AND (NOT "DB7217_TRADES_CALL".GENERAL_CONDITIONS OR NOT "DB7217_TRADES_CALL".CANCEL_2_REQ);
   "DB426_ALARMS_WARNINGS".WARNINGS."743681" := "DB7217_TRADES_CALL".CALL_2;
END_REGION

REGION Network 17: CALL 2 ACKNOWLEDGE
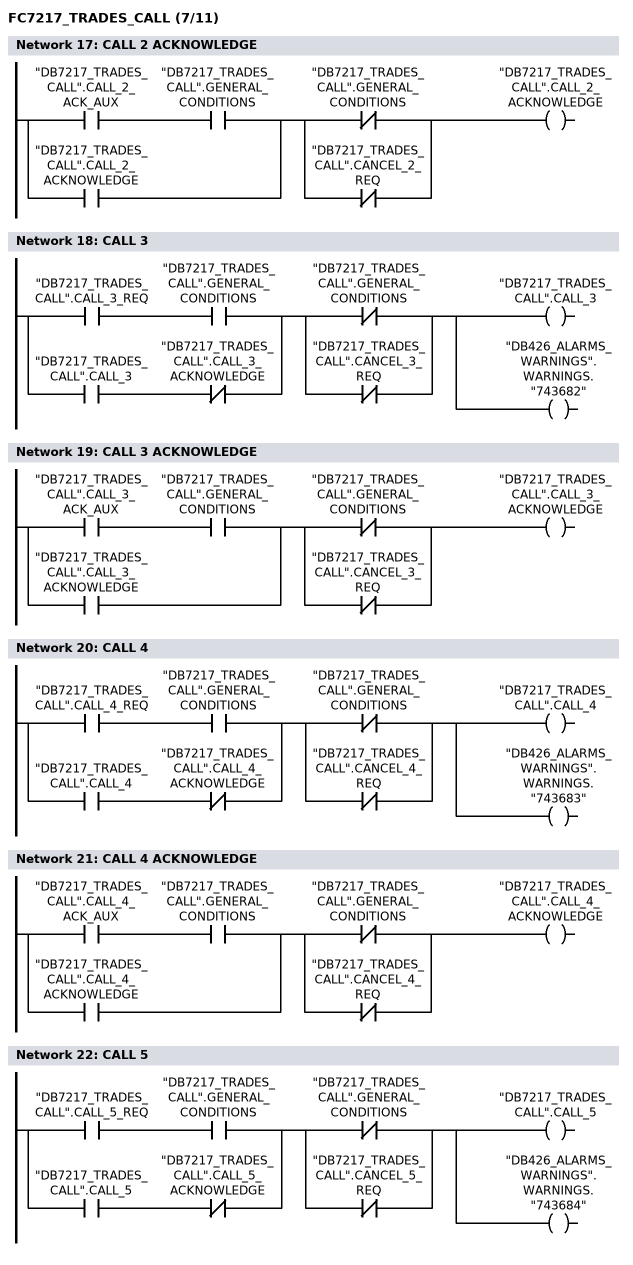
   RUNG wire#powerrail
      Contact( "DB7217_TRADES_CALL".CALL_2_ACK_AUX )
      Contact( "DB7217_TRADES_CALL".GENERAL_CONDITIONS )
      wire#w1
      I_Contact( "DB7217_TRADES_CALL".GENERAL_CONDITIONS )
      wire#w2
      Coil( "DB7217_TRADES_CALL".CALL_2_ACKNOWLEDGE )
   END_RUNG
   RUNG wire#powerrail
      Contact( "DB7217_TRADES_CALL".CALL_2_ACKNOWLEDGE )
   END_RUNG wire#w1
   RUNG wire#w1
      I_Contact( "DB7217_TRADES_CALL".CANCEL_2_REQ )
   END_RUNG wire#w2
   // the same network as SCL:
   "DB7217_TRADES_CALL".CALL_2_ACKNOWLEDGE := (("DB7217_TRADES_CALL".CALL_2_ACK_AUX AND "DB7217_TRADES_CALL".GENERAL_CONDITIONS) OR "DB7217_TRADES_CALL".CALL_2_ACKNOWLEDGE) AND (NOT "DB7217_TRADES_CALL".GENERAL_CONDITIONS OR NOT "DB7217_TRADES_CALL".CANCEL_2_REQ);
END_REGION

REGION Network 18: CALL 3
   RUNG wire#powerrail
      Contact( "DB7217_TRADES_CALL".CALL_3_REQ )
      Contact( "DB7217_TRADES_CALL".GENERAL_CONDITIONS )
      wire#w1
      I_Contact( "DB7217_TRADES_CALL".GENERAL_CONDITIONS )
      wire#w2
      Coil( "DB7217_TRADES_CALL".CALL_3 )
   END_RUNG
   RUNG wire#powerrail
      Contact( "DB7217_TRADES_CALL".CALL_3 )
      I_Contact( "DB7217_TRADES_CALL".CALL_3_ACKNOWLEDGE )
   END_RUNG wire#w1
   RUNG wire#w1
      I_Contact( "DB7217_TRADES_CALL".CANCEL_3_REQ )
   END_RUNG wire#w2
   RUNG wire#w2
      Coil( "DB426_ALARMS_WARNINGS".WARNINGS."743682" )
   END_RUNG
   // the same network as SCL:
   "DB7217_TRADES_CALL".CALL_3 := (("DB7217_TRADES_CALL".CALL_3_REQ AND "DB7217_TRADES_CALL".GENERAL_CONDITIONS) OR ("DB7217_TRADES_CALL".CALL_3 AND NOT "DB7217_TRADES_CALL".CALL_3_ACKNOWLEDGE)) AND (NOT "DB7217_TRADES_CALL".GENERAL_CONDITIONS OR NOT "DB7217_TRADES_CALL".CANCEL_3_REQ);
   "DB426_ALARMS_WARNINGS".WARNINGS."743682" := "DB7217_TRADES_CALL".CALL_3;
END_REGION

REGION Network 19: CALL 3 ACKNOWLEDGE
   RUNG wire#powerrail
      Contact( "DB7217_TRADES_CALL".CALL_3_ACK_AUX )
      Contact( "DB7217_TRADES_CALL".GENERAL_CONDITIONS )
      wire#w1
      I_Contact( "DB7217_TRADES_CALL".GENERAL_CONDITIONS )
      wire#w2
      Coil( "DB7217_TRADES_CALL".CALL_3_ACKNOWLEDGE )
   END_RUNG
   RUNG wire#powerrail
      Contact( "DB7217_TRADES_CALL".CALL_3_ACKNOWLEDGE )
   END_RUNG wire#w1
   RUNG wire#w1
      I_Contact( "DB7217_TRADES_CALL".CANCEL_3_REQ )
   END_RUNG wire#w2
   // the same network as SCL:
   "DB7217_TRADES_CALL".CALL_3_ACKNOWLEDGE := (("DB7217_TRADES_CALL".CALL_3_ACK_AUX AND "DB7217_TRADES_CALL".GENERAL_CONDITIONS) OR "DB7217_TRADES_CALL".CALL_3_ACKNOWLEDGE) AND (NOT "DB7217_TRADES_CALL".GENERAL_CONDITIONS OR NOT "DB7217_TRADES_CALL".CANCEL_3_REQ);
END_REGION

REGION Network 20: CALL 4
   RUNG wire#powerrail
      Contact( "DB7217_TRADES_CALL".CALL_4_REQ )
      Contact( "DB7217_TRADES_CALL".GENERAL_CONDITIONS )
      wire#w1
      I_Contact( "DB7217_TRADES_CALL".GENERAL_CONDITIONS )
      wire#w2
      Coil( "DB7217_TRADES_CALL".CALL_4 )
   END_RUNG
   RUNG wire#powerrail
      Contact( "DB7217_TRADES_CALL".CALL_4 )
      I_Contact( "DB7217_TRADES_CALL".CALL_4_ACKNOWLEDGE )
   END_RUNG wire#w1
   RUNG wire#w1
      I_Contact( "DB7217_TRADES_CALL".CANCEL_4_REQ )
   END_RUNG wire#w2
   RUNG wire#w2
      Coil( "DB426_ALARMS_WARNINGS".WARNINGS."743683" )
   END_RUNG
   // the same network as SCL:
   "DB7217_TRADES_CALL".CALL_4 := (("DB7217_TRADES_CALL".CALL_4_REQ AND "DB7217_TRADES_CALL".GENERAL_CONDITIONS) OR ("DB7217_TRADES_CALL".CALL_4 AND NOT "DB7217_TRADES_CALL".CALL_4_ACKNOWLEDGE)) AND (NOT "DB7217_TRADES_CALL".GENERAL_CONDITIONS OR NOT "DB7217_TRADES_CALL".CANCEL_4_REQ);
   "DB426_ALARMS_WARNINGS".WARNINGS."743683" := "DB7217_TRADES_CALL".CALL_4;
END_REGION

REGION Network 21: CALL 4 ACKNOWLEDGE
   RUNG wire#powerrail
      Contact( "DB7217_TRADES_CALL".CALL_4_ACK_AUX )
      Contact( "DB7217_TRADES_CALL".GENERAL_CONDITIONS )
      wire#w1
      I_Contact( "DB7217_TRADES_CALL".GENERAL_CONDITIONS )
      wire#w2
      Coil( "DB7217_TRADES_CALL".CALL_4_ACKNOWLEDGE )
   END_RUNG
   RUNG wire#powerrail
      Contact( "DB7217_TRADES_CALL".CALL_4_ACKNOWLEDGE )
   END_RUNG wire#w1
   RUNG wire#w1
      I_Contact( "DB7217_TRADES_CALL".CANCEL_4_REQ )
   END_RUNG wire#w2
   // the same network as SCL:
   "DB7217_TRADES_CALL".CALL_4_ACKNOWLEDGE := (("DB7217_TRADES_CALL".CALL_4_ACK_AUX AND "DB7217_TRADES_CALL".GENERAL_CONDITIONS) OR "DB7217_TRADES_CALL".CALL_4_ACKNOWLEDGE) AND (NOT "DB7217_TRADES_CALL".GENERAL_CONDITIONS OR NOT "DB7217_TRADES_CALL".CANCEL_4_REQ);
END_REGION

REGION Network 22: CALL 5
   RUNG wire#powerrail
      Contact( "DB7217_TRADES_CALL".CALL_5_REQ )
      Contact( "DB7217_TRADES_CALL".GENERAL_CONDITIONS )
      wire#w1
      I_Contact( "DB7217_TRADES_CALL".GENERAL_CONDITIONS )
      wire#w2
      Coil( "DB7217_TRADES_CALL".CALL_5 )
   END_RUNG
   RUNG wire#powerrail
      Contact( "DB7217_TRADES_CALL".CALL_5 )
      I_Contact( "DB7217_TRADES_CALL".CALL_5_ACKNOWLEDGE )
   END_RUNG wire#w1
   RUNG wire#w1
      I_Contact( "DB7217_TRADES_CALL".CANCEL_5_REQ )
   END_RUNG wire#w2
   RUNG wire#w2
      Coil( "DB426_ALARMS_WARNINGS".WARNINGS."743684" )
   END_RUNG
   // the same network as SCL:
   "DB7217_TRADES_CALL".CALL_5 := (("DB7217_TRADES_CALL".CALL_5_REQ AND "DB7217_TRADES_CALL".GENERAL_CONDITIONS) OR ("DB7217_TRADES_CALL".CALL_5 AND NOT "DB7217_TRADES_CALL".CALL_5_ACKNOWLEDGE)) AND (NOT "DB7217_TRADES_CALL".GENERAL_CONDITIONS OR NOT "DB7217_TRADES_CALL".CANCEL_5_REQ);
   "DB426_ALARMS_WARNINGS".WARNINGS."743684" := "DB7217_TRADES_CALL".CALL_5;
END_REGION

REGION Network 23: CALL 5 ACKNOWLEDGE
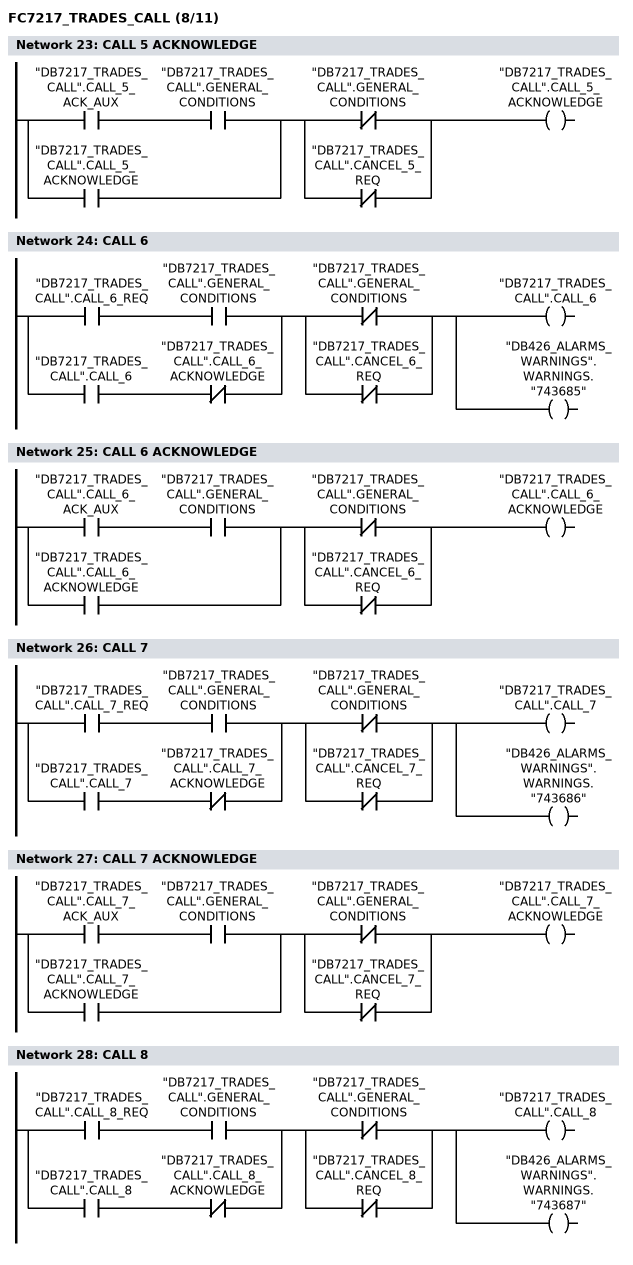
   RUNG wire#powerrail
      Contact( "DB7217_TRADES_CALL".CALL_5_ACK_AUX )
      Contact( "DB7217_TRADES_CALL".GENERAL_CONDITIONS )
      wire#w1
      I_Contact( "DB7217_TRADES_CALL".GENERAL_CONDITIONS )
      wire#w2
      Coil( "DB7217_TRADES_CALL".CALL_5_ACKNOWLEDGE )
   END_RUNG
   RUNG wire#powerrail
      Contact( "DB7217_TRADES_CALL".CALL_5_ACKNOWLEDGE )
   END_RUNG wire#w1
   RUNG wire#w1
      I_Contact( "DB7217_TRADES_CALL".CANCEL_5_REQ )
   END_RUNG wire#w2
   // the same network as SCL:
   "DB7217_TRADES_CALL".CALL_5_ACKNOWLEDGE := (("DB7217_TRADES_CALL".CALL_5_ACK_AUX AND "DB7217_TRADES_CALL".GENERAL_CONDITIONS) OR "DB7217_TRADES_CALL".CALL_5_ACKNOWLEDGE) AND (NOT "DB7217_TRADES_CALL".GENERAL_CONDITIONS OR NOT "DB7217_TRADES_CALL".CANCEL_5_REQ);
END_REGION

REGION Network 24: CALL 6
   RUNG wire#powerrail
      Contact( "DB7217_TRADES_CALL".CALL_6_REQ )
      Contact( "DB7217_TRADES_CALL".GENERAL_CONDITIONS )
      wire#w1
      I_Contact( "DB7217_TRADES_CALL".GENERAL_CONDITIONS )
      wire#w2
      Coil( "DB7217_TRADES_CALL".CALL_6 )
   END_RUNG
   RUNG wire#powerrail
      Contact( "DB7217_TRADES_CALL".CALL_6 )
      I_Contact( "DB7217_TRADES_CALL".CALL_6_ACKNOWLEDGE )
   END_RUNG wire#w1
   RUNG wire#w1
      I_Contact( "DB7217_TRADES_CALL".CANCEL_6_REQ )
   END_RUNG wire#w2
   RUNG wire#w2
      Coil( "DB426_ALARMS_WARNINGS".WARNINGS."743685" )
   END_RUNG
   // the same network as SCL:
   "DB7217_TRADES_CALL".CALL_6 := (("DB7217_TRADES_CALL".CALL_6_REQ AND "DB7217_TRADES_CALL".GENERAL_CONDITIONS) OR ("DB7217_TRADES_CALL".CALL_6 AND NOT "DB7217_TRADES_CALL".CALL_6_ACKNOWLEDGE)) AND (NOT "DB7217_TRADES_CALL".GENERAL_CONDITIONS OR NOT "DB7217_TRADES_CALL".CANCEL_6_REQ);
   "DB426_ALARMS_WARNINGS".WARNINGS."743685" := "DB7217_TRADES_CALL".CALL_6;
END_REGION

REGION Network 25: CALL 6 ACKNOWLEDGE
   RUNG wire#powerrail
      Contact( "DB7217_TRADES_CALL".CALL_6_ACK_AUX )
      Contact( "DB7217_TRADES_CALL".GENERAL_CONDITIONS )
      wire#w1
      I_Contact( "DB7217_TRADES_CALL".GENERAL_CONDITIONS )
      wire#w2
      Coil( "DB7217_TRADES_CALL".CALL_6_ACKNOWLEDGE )
   END_RUNG
   RUNG wire#powerrail
      Contact( "DB7217_TRADES_CALL".CALL_6_ACKNOWLEDGE )
   END_RUNG wire#w1
   RUNG wire#w1
      I_Contact( "DB7217_TRADES_CALL".CANCEL_6_REQ )
   END_RUNG wire#w2
   // the same network as SCL:
   "DB7217_TRADES_CALL".CALL_6_ACKNOWLEDGE := (("DB7217_TRADES_CALL".CALL_6_ACK_AUX AND "DB7217_TRADES_CALL".GENERAL_CONDITIONS) OR "DB7217_TRADES_CALL".CALL_6_ACKNOWLEDGE) AND (NOT "DB7217_TRADES_CALL".GENERAL_CONDITIONS OR NOT "DB7217_TRADES_CALL".CANCEL_6_REQ);
END_REGION

REGION Network 26: CALL 7
   RUNG wire#powerrail
      Contact( "DB7217_TRADES_CALL".CALL_7_REQ )
      Contact( "DB7217_TRADES_CALL".GENERAL_CONDITIONS )
      wire#w1
      I_Contact( "DB7217_TRADES_CALL".GENERAL_CONDITIONS )
      wire#w2
      Coil( "DB7217_TRADES_CALL".CALL_7 )
   END_RUNG
   RUNG wire#powerrail
      Contact( "DB7217_TRADES_CALL".CALL_7 )
      I_Contact( "DB7217_TRADES_CALL".CALL_7_ACKNOWLEDGE )
   END_RUNG wire#w1
   RUNG wire#w1
      I_Contact( "DB7217_TRADES_CALL".CANCEL_7_REQ )
   END_RUNG wire#w2
   RUNG wire#w2
      Coil( "DB426_ALARMS_WARNINGS".WARNINGS."743686" )
   END_RUNG
   // the same network as SCL:
   "DB7217_TRADES_CALL".CALL_7 := (("DB7217_TRADES_CALL".CALL_7_REQ AND "DB7217_TRADES_CALL".GENERAL_CONDITIONS) OR ("DB7217_TRADES_CALL".CALL_7 AND NOT "DB7217_TRADES_CALL".CALL_7_ACKNOWLEDGE)) AND (NOT "DB7217_TRADES_CALL".GENERAL_CONDITIONS OR NOT "DB7217_TRADES_CALL".CANCEL_7_REQ);
   "DB426_ALARMS_WARNINGS".WARNINGS."743686" := "DB7217_TRADES_CALL".CALL_7;
END_REGION

REGION Network 27: CALL 7 ACKNOWLEDGE
   RUNG wire#powerrail
      Contact( "DB7217_TRADES_CALL".CALL_7_ACK_AUX )
      Contact( "DB7217_TRADES_CALL".GENERAL_CONDITIONS )
      wire#w1
      I_Contact( "DB7217_TRADES_CALL".GENERAL_CONDITIONS )
      wire#w2
      Coil( "DB7217_TRADES_CALL".CALL_7_ACKNOWLEDGE )
   END_RUNG
   RUNG wire#powerrail
      Contact( "DB7217_TRADES_CALL".CALL_7_ACKNOWLEDGE )
   END_RUNG wire#w1
   RUNG wire#w1
      I_Contact( "DB7217_TRADES_CALL".CANCEL_7_REQ )
   END_RUNG wire#w2
   // the same network as SCL:
   "DB7217_TRADES_CALL".CALL_7_ACKNOWLEDGE := (("DB7217_TRADES_CALL".CALL_7_ACK_AUX AND "DB7217_TRADES_CALL".GENERAL_CONDITIONS) OR "DB7217_TRADES_CALL".CALL_7_ACKNOWLEDGE) AND (NOT "DB7217_TRADES_CALL".GENERAL_CONDITIONS OR NOT "DB7217_TRADES_CALL".CANCEL_7_REQ);
END_REGION

REGION Network 28: CALL 8
   RUNG wire#powerrail
      Contact( "DB7217_TRADES_CALL".CALL_8_REQ )
      Contact( "DB7217_TRADES_CALL".GENERAL_CONDITIONS )
      wire#w1
      I_Contact( "DB7217_TRADES_CALL".GENERAL_CONDITIONS )
      wire#w2
      Coil( "DB7217_TRADES_CALL".CALL_8 )
   END_RUNG
   RUNG wire#powerrail
      Contact( "DB7217_TRADES_CALL".CALL_8 )
      I_Contact( "DB7217_TRADES_CALL".CALL_8_ACKNOWLEDGE )
   END_RUNG wire#w1
   RUNG wire#w1
      I_Contact( "DB7217_TRADES_CALL".CANCEL_8_REQ )
   END_RUNG wire#w2
   RUNG wire#w2
      Coil( "DB426_ALARMS_WARNINGS".WARNINGS."743687" )
   END_RUNG
   // the same network as SCL:
   "DB7217_TRADES_CALL".CALL_8 := (("DB7217_TRADES_CALL".CALL_8_REQ AND "DB7217_TRADES_CALL".GENERAL_CONDITIONS) OR ("DB7217_TRADES_CALL".CALL_8 AND NOT "DB7217_TRADES_CALL".CALL_8_ACKNOWLEDGE)) AND (NOT "DB7217_TRADES_CALL".GENERAL_CONDITIONS OR NOT "DB7217_TRADES_CALL".CANCEL_8_REQ);
   "DB426_ALARMS_WARNINGS".WARNINGS."743687" := "DB7217_TRADES_CALL".CALL_8;
END_REGION

REGION Network 29: CALL 8 ACKNOWLEDGE
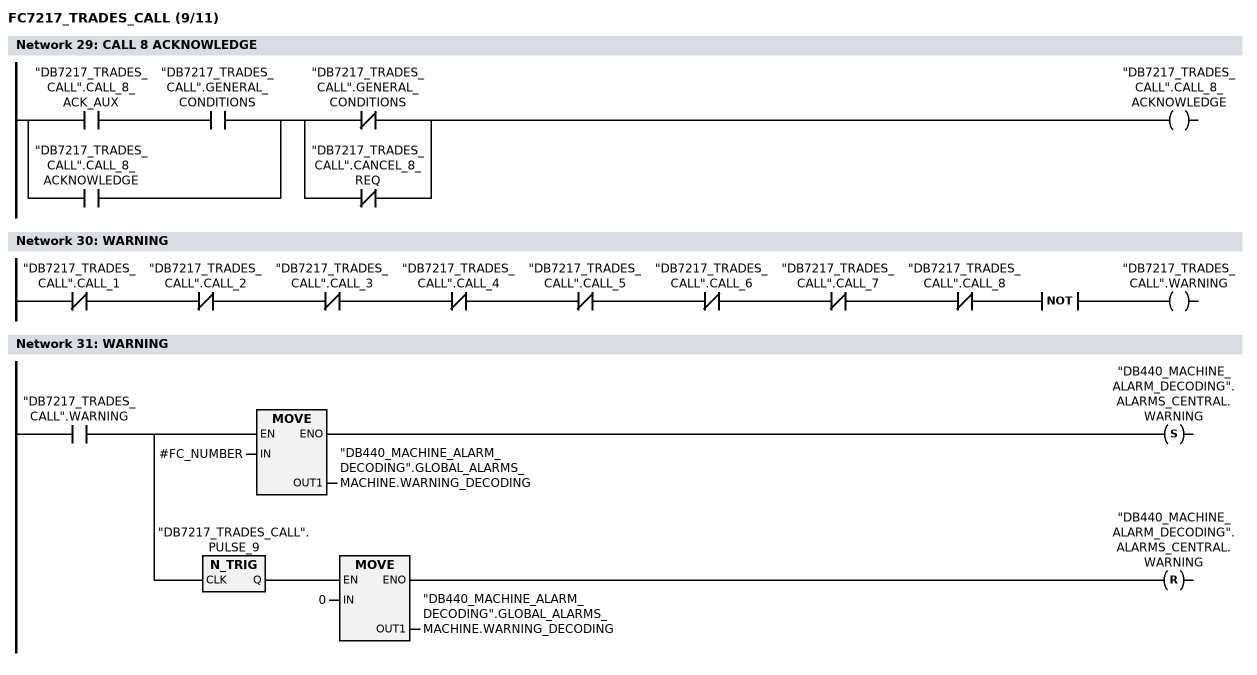
   RUNG wire#powerrail
      Contact( "DB7217_TRADES_CALL".CALL_8_ACK_AUX )
      Contact( "DB7217_TRADES_CALL".GENERAL_CONDITIONS )
      wire#w1
      I_Contact( "DB7217_TRADES_CALL".GENERAL_CONDITIONS )
      wire#w2
      Coil( "DB7217_TRADES_CALL".CALL_8_ACKNOWLEDGE )
   END_RUNG
   RUNG wire#powerrail
      Contact( "DB7217_TRADES_CALL".CALL_8_ACKNOWLEDGE )
   END_RUNG wire#w1
   RUNG wire#w1
      I_Contact( "DB7217_TRADES_CALL".CANCEL_8_REQ )
   END_RUNG wire#w2
   // the same network as SCL:
   "DB7217_TRADES_CALL".CALL_8_ACKNOWLEDGE := (("DB7217_TRADES_CALL".CALL_8_ACK_AUX AND "DB7217_TRADES_CALL".GENERAL_CONDITIONS) OR "DB7217_TRADES_CALL".CALL_8_ACKNOWLEDGE) AND (NOT "DB7217_TRADES_CALL".GENERAL_CONDITIONS OR NOT "DB7217_TRADES_CALL".CANCEL_8_REQ);
END_REGION

REGION Network 30: WARNING
   RUNG wire#powerrail
      I_Contact( "DB7217_TRADES_CALL".CALL_1 )
      I_Contact( "DB7217_TRADES_CALL".CALL_2 )
      I_Contact( "DB7217_TRADES_CALL".CALL_3 )
      I_Contact( "DB7217_TRADES_CALL".CALL_4 )
      I_Contact( "DB7217_TRADES_CALL".CALL_5 )
      I_Contact( "DB7217_TRADES_CALL".CALL_6 )
      I_Contact( "DB7217_TRADES_CALL".CALL_7 )
      I_Contact( "DB7217_TRADES_CALL".CALL_8 )
      Not()
      Coil( "DB7217_TRADES_CALL".WARNING )
   END_RUNG
   // the same network as SCL:
   "DB7217_TRADES_CALL".WARNING := NOT (NOT "DB7217_TRADES_CALL".CALL_1 AND NOT "DB7217_TRADES_CALL".CALL_2 AND NOT "DB7217_TRADES_CALL".CALL_3 AND NOT "DB7217_TRADES_CALL".CALL_4 AND NOT "DB7217_TRADES_CALL".CALL_5 AND NOT "DB7217_TRADES_CALL".CALL_6 AND NOT "DB7217_TRADES_CALL".CALL_7 AND NOT "DB7217_TRADES_CALL".CALL_8);
END_REGION

REGION Network 31: WARNING
   RUNG wire#powerrail
      Contact( "DB7217_TRADES_CALL".WARNING )
      wire#w1
      { S7_GenerateENO := "TRUE" } Move(in := #FC_NUMBER, out1 => "DB440_MACHINE_ALARM_DECODING".GLOBAL_ALARMS_MACHINE.WARNING_DECODING)
      S_Coil( "DB440_MACHINE_ALARM_DECODING".ALARMS_CENTRAL.WARNING )
   END_RUNG
   RUNG wire#w1
      N_Trig( "DB7217_TRADES_CALL".PULSE_9 )
      { S7_GenerateENO := "TRUE" } Move(in := 0, out1 => "DB440_MACHINE_ALARM_DECODING".GLOBAL_ALARMS_MACHINE.WARNING_DECODING)
      R_Coil( "DB440_MACHINE_ALARM_DECODING".ALARMS_CENTRAL.WARNING )
   END_RUNG
   // the same network as SCL:
   // ENO of a box is taken as its EN; it also drops when the box reports an error
   IF "DB7217_TRADES_CALL".WARNING THEN
       "DB440_MACHINE_ALARM_DECODING".GLOBAL_ALARMS_MACHINE.WARNING_DECODING := #FC_NUMBER;
       "DB440_MACHINE_ALARM_DECODING".ALARMS_CENTRAL.WARNING := TRUE;
   END_IF;
   #_w1 := NOT "DB7217_TRADES_CALL".WARNING AND "DB7217_TRADES_CALL".PULSE_9;   // falling edge
   "DB7217_TRADES_CALL".PULSE_9 := "DB7217_TRADES_CALL".WARNING;
   IF #_w1 THEN
       "DB440_MACHINE_ALARM_DECODING".GLOBAL_ALARMS_MACHINE.WARNING_DECODING := 0;
       "DB440_MACHINE_ALARM_DECODING".ALARMS_CENTRAL.WARNING := FALSE;
   END_IF;
END_REGION

REGION Network 32: HMI STATUS
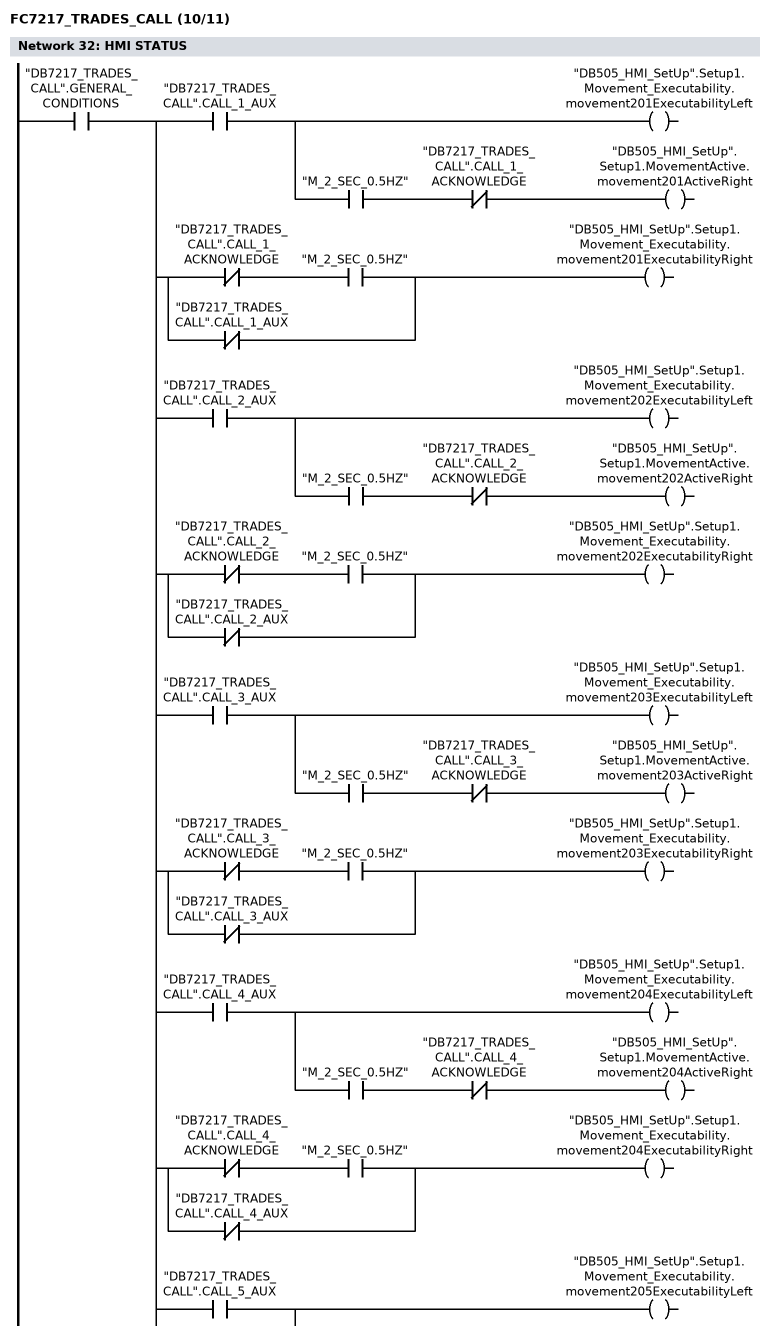
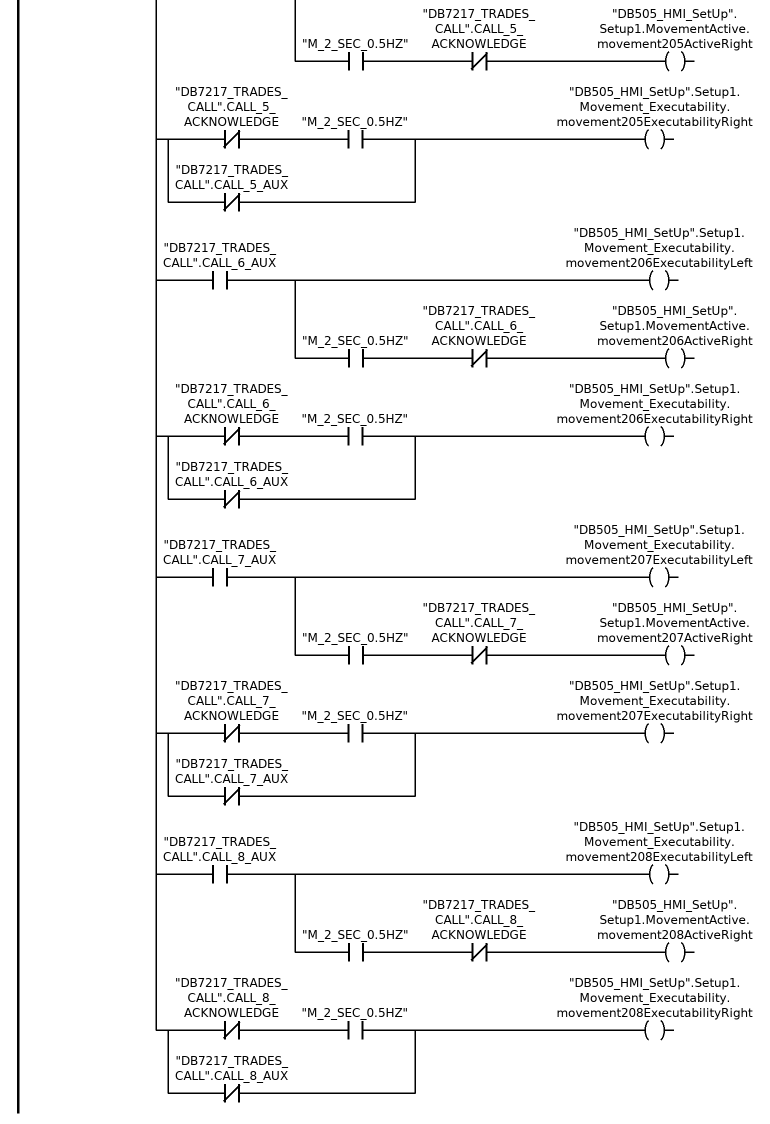
   RUNG wire#powerrail
      Contact( "DB7217_TRADES_CALL".GENERAL_CONDITIONS )
      wire#w1
      Contact( "DB7217_TRADES_CALL".CALL_1_AUX )
      wire#w2
      Coil( "DB505_HMI_SetUp".Setup1.Movement_Executability.movement201ExecutabilityLeft )
   END_RUNG
   RUNG wire#w2
      Contact( "M_2_SEC_0.5HZ" )
      I_Contact( "DB7217_TRADES_CALL".CALL_1_ACKNOWLEDGE )
      Coil( "DB505_HMI_SetUp".Setup1.MovementActive.movement201ActiveRight )
   END_RUNG
   RUNG wire#w1
      I_Contact( "DB7217_TRADES_CALL".CALL_1_ACKNOWLEDGE )
      Contact( "M_2_SEC_0.5HZ" )
      wire#w3
      Coil( "DB505_HMI_SetUp".Setup1.Movement_Executability.movement201ExecutabilityRight )
   END_RUNG
   RUNG wire#w1
      I_Contact( "DB7217_TRADES_CALL".CALL_1_AUX )
   END_RUNG wire#w3
   RUNG wire#w1
      Contact( "DB7217_TRADES_CALL".CALL_2_AUX )
      wire#w4
      Coil( "DB505_HMI_SetUp".Setup1.Movement_Executability.movement202ExecutabilityLeft )
   END_RUNG
   RUNG wire#w4
      Contact( "M_2_SEC_0.5HZ" )
      I_Contact( "DB7217_TRADES_CALL".CALL_2_ACKNOWLEDGE )
      Coil( "DB505_HMI_SetUp".Setup1.MovementActive.movement202ActiveRight )
   END_RUNG
   RUNG wire#w1
      I_Contact( "DB7217_TRADES_CALL".CALL_2_ACKNOWLEDGE )
      Contact( "M_2_SEC_0.5HZ" )
      wire#w5
      Coil( "DB505_HMI_SetUp".Setup1.Movement_Executability.movement202ExecutabilityRight )
   END_RUNG
   RUNG wire#w1
      I_Contact( "DB7217_TRADES_CALL".CALL_2_AUX )
   END_RUNG wire#w5
   RUNG wire#w1
      Contact( "DB7217_TRADES_CALL".CALL_3_AUX )
      wire#w6
      Coil( "DB505_HMI_SetUp".Setup1.Movement_Executability.movement203ExecutabilityLeft )
   END_RUNG
   RUNG wire#w6
      Contact( "M_2_SEC_0.5HZ" )
      I_Contact( "DB7217_TRADES_CALL".CALL_3_ACKNOWLEDGE )
      Coil( "DB505_HMI_SetUp".Setup1.MovementActive.movement203ActiveRight )
   END_RUNG
   RUNG wire#w1
      I_Contact( "DB7217_TRADES_CALL".CALL_3_ACKNOWLEDGE )
      Contact( "M_2_SEC_0.5HZ" )
      wire#w7
      Coil( "DB505_HMI_SetUp".Setup1.Movement_Executability.movement203ExecutabilityRight )
   END_RUNG
   RUNG wire#w1
      I_Contact( "DB7217_TRADES_CALL".CALL_3_AUX )
   END_RUNG wire#w7
   RUNG wire#w1
      Contact( "DB7217_TRADES_CALL".CALL_4_AUX )
      wire#w8
      Coil( "DB505_HMI_SetUp".Setup1.Movement_Executability.movement204ExecutabilityLeft )
   END_RUNG
   RUNG wire#w8
      Contact( "M_2_SEC_0.5HZ" )
      I_Contact( "DB7217_TRADES_CALL".CALL_4_ACKNOWLEDGE )
      Coil( "DB505_HMI_SetUp".Setup1.MovementActive.movement204ActiveRight )
   END_RUNG
   RUNG wire#w1
      I_Contact( "DB7217_TRADES_CALL".CALL_4_ACKNOWLEDGE )
      Contact( "M_2_SEC_0.5HZ" )
      wire#w9
      Coil( "DB505_HMI_SetUp".Setup1.Movement_Executability.movement204ExecutabilityRight )
   END_RUNG
   RUNG wire#w1
      I_Contact( "DB7217_TRADES_CALL".CALL_4_AUX )
   END_RUNG wire#w9
   RUNG wire#w1
      Contact( "DB7217_TRADES_CALL".CALL_5_AUX )
      wire#w10
      Coil( "DB505_HMI_SetUp".Setup1.Movement_Executability.movement205ExecutabilityLeft )
   END_RUNG
   RUNG wire#w10
      Contact( "M_2_SEC_0.5HZ" )
      I_Contact( "DB7217_TRADES_CALL".CALL_5_ACKNOWLEDGE )
      Coil( "DB505_HMI_SetUp".Setup1.MovementActive.movement205ActiveRight )
   END_RUNG
   RUNG wire#w1
      I_Contact( "DB7217_TRADES_CALL".CALL_5_ACKNOWLEDGE )
      Contact( "M_2_SEC_0.5HZ" )
      wire#w11
      Coil( "DB505_HMI_SetUp".Setup1.Movement_Executability.movement205ExecutabilityRight )
   END_RUNG
   RUNG wire#w1
      I_Contact( "DB7217_TRADES_CALL".CALL_5_AUX )
   END_RUNG wire#w11
   RUNG wire#w1
      Contact( "DB7217_TRADES_CALL".CALL_6_AUX )
      wire#w12
      Coil( "DB505_HMI_SetUp".Setup1.Movement_Executability.movement206ExecutabilityLeft )
   END_RUNG
   RUNG wire#w12
      Contact( "M_2_SEC_0.5HZ" )
      I_Contact( "DB7217_TRADES_CALL".CALL_6_ACKNOWLEDGE )
      Coil( "DB505_HMI_SetUp".Setup1.MovementActive.movement206ActiveRight )
   END_RUNG
   RUNG wire#w1
      I_Contact( "DB7217_TRADES_CALL".CALL_6_ACKNOWLEDGE )
      Contact( "M_2_SEC_0.5HZ" )
      wire#w13
      Coil( "DB505_HMI_SetUp".Setup1.Movement_Executability.movement206ExecutabilityRight )
   END_RUNG
   RUNG wire#w1
      I_Contact( "DB7217_TRADES_CALL".CALL_6_AUX )
   END_RUNG wire#w13
   RUNG wire#w1
      Contact( "DB7217_TRADES_CALL".CALL_7_AUX )
      wire#w14
      Coil( "DB505_HMI_SetUp".Setup1.Movement_Executability.movement207ExecutabilityLeft )
   END_RUNG
   RUNG wire#w14
      Contact( "M_2_SEC_0.5HZ" )
      I_Contact( "DB7217_TRADES_CALL".CALL_7_ACKNOWLEDGE )
      Coil( "DB505_HMI_SetUp".Setup1.MovementActive.movement207ActiveRight )
   END_RUNG
   RUNG wire#w1
      I_Contact( "DB7217_TRADES_CALL".CALL_7_ACKNOWLEDGE )
      Contact( "M_2_SEC_0.5HZ" )
      wire#w15
      Coil( "DB505_HMI_SetUp".Setup1.Movement_Executability.movement207ExecutabilityRight )
   END_RUNG
   RUNG wire#w1
      I_Contact( "DB7217_TRADES_CALL".CALL_7_AUX )
   END_RUNG wire#w15
   RUNG wire#w1
      Contact( "DB7217_TRADES_CALL".CALL_8_AUX )
      wire#w16
      Coil( "DB505_HMI_SetUp".Setup1.Movement_Executability.movement208ExecutabilityLeft )
   END_RUNG
   RUNG wire#w16
      Contact( "M_2_SEC_0.5HZ" )
      I_Contact( "DB7217_TRADES_CALL".CALL_8_ACKNOWLEDGE )
      Coil( "DB505_HMI_SetUp".Setup1.MovementActive.movement208ActiveRight )
   END_RUNG
   RUNG wire#w1
      I_Contact( "DB7217_TRADES_CALL".CALL_8_ACKNOWLEDGE )
      Contact( "M_2_SEC_0.5HZ" )
      wire#w17
      Coil( "DB505_HMI_SetUp".Setup1.Movement_Executability.movement208ExecutabilityRight )
   END_RUNG
   RUNG wire#w1
      I_Contact( "DB7217_TRADES_CALL".CALL_8_AUX )
   END_RUNG wire#w17
   // the same network as SCL:
   "DB505_HMI_SetUp".Setup1.Movement_Executability.movement201ExecutabilityLeft := "DB7217_TRADES_CALL".GENERAL_CONDITIONS AND "DB7217_TRADES_CALL".CALL_1_AUX;
   "DB505_HMI_SetUp".Setup1.MovementActive.movement201ActiveRight := "DB505_HMI_SetUp".Setup1.Movement_Executability.movement201ExecutabilityLeft AND "M_2_SEC_0.5HZ" AND NOT "DB7217_TRADES_CALL".CALL_1_ACKNOWLEDGE;
   "DB505_HMI_SetUp".Setup1.Movement_Executability.movement201ExecutabilityRight := "DB7217_TRADES_CALL".GENERAL_CONDITIONS AND ((NOT "DB7217_TRADES_CALL".CALL_1_ACKNOWLEDGE AND "M_2_SEC_0.5HZ") OR NOT "DB7217_TRADES_CALL".CALL_1_AUX);
   "DB505_HMI_SetUp".Setup1.Movement_Executability.movement202ExecutabilityLeft := "DB7217_TRADES_CALL".GENERAL_CONDITIONS AND "DB7217_TRADES_CALL".CALL_2_AUX;
   "DB505_HMI_SetUp".Setup1.MovementActive.movement202ActiveRight := "DB505_HMI_SetUp".Setup1.Movement_Executability.movement202ExecutabilityLeft AND "M_2_SEC_0.5HZ" AND NOT "DB7217_TRADES_CALL".CALL_2_ACKNOWLEDGE;
   "DB505_HMI_SetUp".Setup1.Movement_Executability.movement202ExecutabilityRight := "DB7217_TRADES_CALL".GENERAL_CONDITIONS AND ((NOT "DB7217_TRADES_CALL".CALL_2_ACKNOWLEDGE AND "M_2_SEC_0.5HZ") OR NOT "DB7217_TRADES_CALL".CALL_2_AUX);
   "DB505_HMI_SetUp".Setup1.Movement_Executability.movement203ExecutabilityLeft := "DB7217_TRADES_CALL".GENERAL_CONDITIONS AND "DB7217_TRADES_CALL".CALL_3_AUX;
   "DB505_HMI_SetUp".Setup1.MovementActive.movement203ActiveRight := "DB505_HMI_SetUp".Setup1.Movement_Executability.movement203ExecutabilityLeft AND "M_2_SEC_0.5HZ" AND NOT "DB7217_TRADES_CALL".CALL_3_ACKNOWLEDGE;
   "DB505_HMI_SetUp".Setup1.Movement_Executability.movement203ExecutabilityRight := "DB7217_TRADES_CALL".GENERAL_CONDITIONS AND ((NOT "DB7217_TRADES_CALL".CALL_3_ACKNOWLEDGE AND "M_2_SEC_0.5HZ") OR NOT "DB7217_TRADES_CALL".CALL_3_AUX);
   "DB505_HMI_SetUp".Setup1.Movement_Executability.movement204ExecutabilityLeft := "DB7217_TRADES_CALL".GENERAL_CONDITIONS AND "DB7217_TRADES_CALL".CALL_4_AUX;
   "DB505_HMI_SetUp".Setup1.MovementActive.movement204ActiveRight := "DB505_HMI_SetUp".Setup1.Movement_Executability.movement204ExecutabilityLeft AND "M_2_SEC_0.5HZ" AND NOT "DB7217_TRADES_CALL".CALL_4_ACKNOWLEDGE;
   "DB505_HMI_SetUp".Setup1.Movement_Executability.movement204ExecutabilityRight := "DB7217_TRADES_CALL".GENERAL_CONDITIONS AND ((NOT "DB7217_TRADES_CALL".CALL_4_ACKNOWLEDGE AND "M_2_SEC_0.5HZ") OR NOT "DB7217_TRADES_CALL".CALL_4_AUX);
   "DB505_HMI_SetUp".Setup1.Movement_Executability.movement205ExecutabilityLeft := "DB7217_TRADES_CALL".GENERAL_CONDITIONS AND "DB7217_TRADES_CALL".CALL_5_AUX;
   "DB505_HMI_SetUp".Setup1.MovementActive.movement205ActiveRight := "DB505_HMI_SetUp".Setup1.Movement_Executability.movement205ExecutabilityLeft AND "M_2_SEC_0.5HZ" AND NOT "DB7217_TRADES_CALL".CALL_5_ACKNOWLEDGE;
   "DB505_HMI_SetUp".Setup1.Movement_Executability.movement205ExecutabilityRight := "DB7217_TRADES_CALL".GENERAL_CONDITIONS AND ((NOT "DB7217_TRADES_CALL".CALL_5_ACKNOWLEDGE AND "M_2_SEC_0.5HZ") OR NOT "DB7217_TRADES_CALL".CALL_5_AUX);
   "DB505_HMI_SetUp".Setup1.Movement_Executability.movement206ExecutabilityLeft := "DB7217_TRADES_CALL".GENERAL_CONDITIONS AND "DB7217_TRADES_CALL".CALL_6_AUX;
   "DB505_HMI_SetUp".Setup1.MovementActive.movement206ActiveRight := "DB505_HMI_SetUp".Setup1.Movement_Executability.movement206ExecutabilityLeft AND "M_2_SEC_0.5HZ" AND NOT "DB7217_TRADES_CALL".CALL_6_ACKNOWLEDGE;
   "DB505_HMI_SetUp".Setup1.Movement_Executability.movement206ExecutabilityRight := "DB7217_TRADES_CALL".GENERAL_CONDITIONS AND ((NOT "DB7217_TRADES_CALL".CALL_6_ACKNOWLEDGE AND "M_2_SEC_0.5HZ") OR NOT "DB7217_TRADES_CALL".CALL_6_AUX);
   "DB505_HMI_SetUp".Setup1.Movement_Executability.movement207ExecutabilityLeft := "DB7217_TRADES_CALL".GENERAL_CONDITIONS AND "DB7217_TRADES_CALL".CALL_7_AUX;
   "DB505_HMI_SetUp".Setup1.MovementActive.movement207ActiveRight := "DB505_HMI_SetUp".Setup1.Movement_Executability.movement207ExecutabilityLeft AND "M_2_SEC_0.5HZ" AND NOT "DB7217_TRADES_CALL".CALL_7_ACKNOWLEDGE;
   "DB505_HMI_SetUp".Setup1.Movement_Executability.movement207ExecutabilityRight := "DB7217_TRADES_CALL".GENERAL_CONDITIONS AND ((NOT "DB7217_TRADES_CALL".CALL_7_ACKNOWLEDGE AND "M_2_SEC_0.5HZ") OR NOT "DB7217_TRADES_CALL".CALL_7_AUX);
   "DB505_HMI_SetUp".Setup1.Movement_Executability.movement208ExecutabilityLeft := "DB7217_TRADES_CALL".GENERAL_CONDITIONS AND "DB7217_TRADES_CALL".CALL_8_AUX;
   "DB505_HMI_SetUp".Setup1.MovementActive.movement208ActiveRight := "DB505_HMI_SetUp".Setup1.Movement_Executability.movement208ExecutabilityLeft AND "M_2_SEC_0.5HZ" AND NOT "DB7217_TRADES_CALL".CALL_8_ACKNOWLEDGE;
   "DB505_HMI_SetUp".Setup1.Movement_Executability.movement208ExecutabilityRight := "DB7217_TRADES_CALL".GENERAL_CONDITIONS AND ((NOT "DB7217_TRADES_CALL".CALL_8_ACKNOWLEDGE AND "M_2_SEC_0.5HZ") OR NOT "DB7217_TRADES_CALL".CALL_8_AUX);
END_REGION

REGION Network 33: HMI STATUS
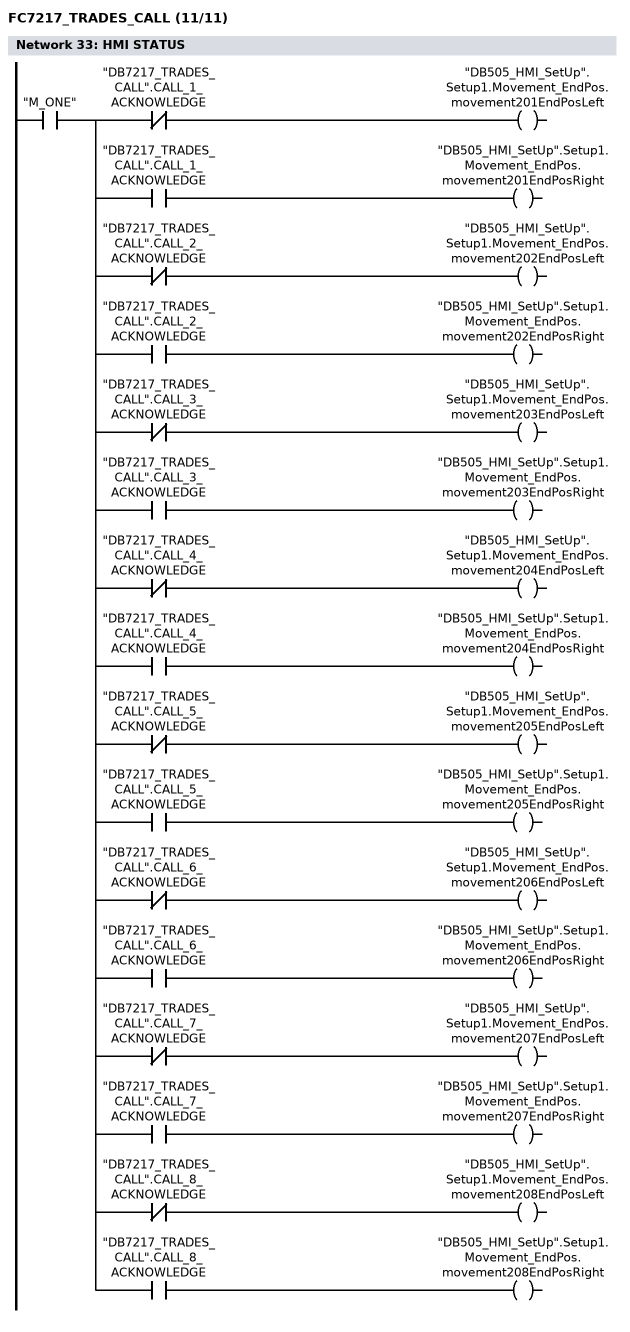
   RUNG wire#powerrail
      Contact( "M_ONE" )
      wire#w1
      I_Contact( "DB7217_TRADES_CALL".CALL_1_ACKNOWLEDGE )
      Coil( "DB505_HMI_SetUp".Setup1.Movement_EndPos.movement201EndPosLeft )
   END_RUNG
   RUNG wire#w1
      Contact( "DB7217_TRADES_CALL".CALL_1_ACKNOWLEDGE )
      Coil( "DB505_HMI_SetUp".Setup1.Movement_EndPos.movement201EndPosRight )
   END_RUNG
   RUNG wire#w1
      I_Contact( "DB7217_TRADES_CALL".CALL_2_ACKNOWLEDGE )
      Coil( "DB505_HMI_SetUp".Setup1.Movement_EndPos.movement202EndPosLeft )
   END_RUNG
   RUNG wire#w1
      Contact( "DB7217_TRADES_CALL".CALL_2_ACKNOWLEDGE )
      Coil( "DB505_HMI_SetUp".Setup1.Movement_EndPos.movement202EndPosRight )
   END_RUNG
   RUNG wire#w1
      I_Contact( "DB7217_TRADES_CALL".CALL_3_ACKNOWLEDGE )
      Coil( "DB505_HMI_SetUp".Setup1.Movement_EndPos.movement203EndPosLeft )
   END_RUNG
   RUNG wire#w1
      Contact( "DB7217_TRADES_CALL".CALL_3_ACKNOWLEDGE )
      Coil( "DB505_HMI_SetUp".Setup1.Movement_EndPos.movement203EndPosRight )
   END_RUNG
   RUNG wire#w1
      I_Contact( "DB7217_TRADES_CALL".CALL_4_ACKNOWLEDGE )
      Coil( "DB505_HMI_SetUp".Setup1.Movement_EndPos.movement204EndPosLeft )
   END_RUNG
   RUNG wire#w1
      Contact( "DB7217_TRADES_CALL".CALL_4_ACKNOWLEDGE )
      Coil( "DB505_HMI_SetUp".Setup1.Movement_EndPos.movement204EndPosRight )
   END_RUNG
   RUNG wire#w1
      I_Contact( "DB7217_TRADES_CALL".CALL_5_ACKNOWLEDGE )
      Coil( "DB505_HMI_SetUp".Setup1.Movement_EndPos.movement205EndPosLeft )
   END_RUNG
   RUNG wire#w1
      Contact( "DB7217_TRADES_CALL".CALL_5_ACKNOWLEDGE )
      Coil( "DB505_HMI_SetUp".Setup1.Movement_EndPos.movement205EndPosRight )
   END_RUNG
   RUNG wire#w1
      I_Contact( "DB7217_TRADES_CALL".CALL_6_ACKNOWLEDGE )
      Coil( "DB505_HMI_SetUp".Setup1.Movement_EndPos.movement206EndPosLeft )
   END_RUNG
   RUNG wire#w1
      Contact( "DB7217_TRADES_CALL".CALL_6_ACKNOWLEDGE )
      Coil( "DB505_HMI_SetUp".Setup1.Movement_EndPos.movement206EndPosRight )
   END_RUNG
   RUNG wire#w1
      I_Contact( "DB7217_TRADES_CALL".CALL_7_ACKNOWLEDGE )
      Coil( "DB505_HMI_SetUp".Setup1.Movement_EndPos.movement207EndPosLeft )
   END_RUNG
   RUNG wire#w1
      Contact( "DB7217_TRADES_CALL".CALL_7_ACKNOWLEDGE )
      Coil( "DB505_HMI_SetUp".Setup1.Movement_EndPos.movement207EndPosRight )
   END_RUNG
   RUNG wire#w1
      I_Contact( "DB7217_TRADES_CALL".CALL_8_ACKNOWLEDGE )
      Coil( "DB505_HMI_SetUp".Setup1.Movement_EndPos.movement208EndPosLeft )
   END_RUNG
   RUNG wire#w1
      Contact( "DB7217_TRADES_CALL".CALL_8_ACKNOWLEDGE )
      Coil( "DB505_HMI_SetUp".Setup1.Movement_EndPos.movement208EndPosRight )
   END_RUNG
   // the same network as SCL:
   "DB505_HMI_SetUp".Setup1.Movement_EndPos.movement201EndPosLeft := "M_ONE" AND NOT "DB7217_TRADES_CALL".CALL_1_ACKNOWLEDGE;
   "DB505_HMI_SetUp".Setup1.Movement_EndPos.movement201EndPosRight := "M_ONE" AND "DB7217_TRADES_CALL".CALL_1_ACKNOWLEDGE;
   "DB505_HMI_SetUp".Setup1.Movement_EndPos.movement202EndPosLeft := "M_ONE" AND NOT "DB7217_TRADES_CALL".CALL_2_ACKNOWLEDGE;
   "DB505_HMI_SetUp".Setup1.Movement_EndPos.movement202EndPosRight := "M_ONE" AND "DB7217_TRADES_CALL".CALL_2_ACKNOWLEDGE;
   "DB505_HMI_SetUp".Setup1.Movement_EndPos.movement203EndPosLeft := "M_ONE" AND NOT "DB7217_TRADES_CALL".CALL_3_ACKNOWLEDGE;
   "DB505_HMI_SetUp".Setup1.Movement_EndPos.movement203EndPosRight := "M_ONE" AND "DB7217_TRADES_CALL".CALL_3_ACKNOWLEDGE;
   "DB505_HMI_SetUp".Setup1.Movement_EndPos.movement204EndPosLeft := "M_ONE" AND NOT "DB7217_TRADES_CALL".CALL_4_ACKNOWLEDGE;
   "DB505_HMI_SetUp".Setup1.Movement_EndPos.movement204EndPosRight := "M_ONE" AND "DB7217_TRADES_CALL".CALL_4_ACKNOWLEDGE;
   "DB505_HMI_SetUp".Setup1.Movement_EndPos.movement205EndPosLeft := "M_ONE" AND NOT "DB7217_TRADES_CALL".CALL_5_ACKNOWLEDGE;
   "DB505_HMI_SetUp".Setup1.Movement_EndPos.movement205EndPosRight := "M_ONE" AND "DB7217_TRADES_CALL".CALL_5_ACKNOWLEDGE;
   "DB505_HMI_SetUp".Setup1.Movement_EndPos.movement206EndPosLeft := "M_ONE" AND NOT "DB7217_TRADES_CALL".CALL_6_ACKNOWLEDGE;
   "DB505_HMI_SetUp".Setup1.Movement_EndPos.movement206EndPosRight := "M_ONE" AND "DB7217_TRADES_CALL".CALL_6_ACKNOWLEDGE;
   "DB505_HMI_SetUp".Setup1.Movement_EndPos.movement207EndPosLeft := "M_ONE" AND NOT "DB7217_TRADES_CALL".CALL_7_ACKNOWLEDGE;
   "DB505_HMI_SetUp".Setup1.Movement_EndPos.movement207EndPosRight := "M_ONE" AND "DB7217_TRADES_CALL".CALL_7_ACKNOWLEDGE;
   "DB505_HMI_SetUp".Setup1.Movement_EndPos.movement208EndPosLeft := "M_ONE" AND NOT "DB7217_TRADES_CALL".CALL_8_ACKNOWLEDGE;
   "DB505_HMI_SetUp".Setup1.Movement_EndPos.movement208EndPosRight := "M_ONE" AND "DB7217_TRADES_CALL".CALL_8_ACKNOWLEDGE;
END_REGION
END_FUNCTION
